   1:  PR[91,1] = PR[90,1] + 52.071;
   1:  PR[91,2] = PR[90,2] + -8.598;
   1:L PR[91] R[100]mm/sec CNT100;
   1:  PR[91,1] = PR[90,1] + 52.540;
   1:  PR[91,2] = PR[90,2] + -9.595;
   1:L PR[91] R[100]mm/sec CNT100;
   1:  PR[91,1] = PR[90,1] + 55.300;
   1:  PR[91,2] = PR[90,2] + -13.179;
   1:L PR[91] R[100]mm/sec CNT100;
   1:  PR[91,1] = PR[90,1] + 55.787;
   1:  PR[91,2] = PR[90,2] + -13.569;
   1:L PR[91] R[100]mm/sec CNT100;
   1:  PR[91,1] = PR[90,1] + 58.893;
   1:  PR[91,2] = PR[90,2] + -16.268;
   1:L PR[91] R[100]mm/sec CNT100;
   1:  PR[91,1] = PR[90,1] + 59.466;
   1:  PR[91,2] = PR[90,2] + -16.585;
   1:L PR[91] R[100]mm/sec CNT100;
   1:  PR[91,1] = PR[90,1] + 62.965;
   1:  PR[91,2] = PR[90,2] + -18.448;
   1:L PR[91] R[100]mm/sec CNT100;
   1:  PR[91,1] = PR[90,1] + 64.665;
   1:  PR[91,2] = PR[90,2] + -18.947;
   1:L PR[91] R[100]mm/sec CNT100;
   1:  PR[91,1] = PR[90,1] + 67.396;
   1:  PR[91,2] = PR[90,2] + -19.702;
   1:L PR[91] R[100]mm/sec CNT100;
   1:  PR[91,1] = PR[90,1] + 70.206;
   1:  PR[91,2] = PR[90,2] + -19.904;
   1:L PR[91] R[100]mm/sec CNT100;
   1:  PR[91,1] = PR[90,1] + 71.961;
   1:  PR[91,2] = PR[90,2] + -20.003;
   1:L PR[91] R[100]mm/sec CNT100;
   1:  PR[91,1] = PR[90,1] + 75.629;
   1:  PR[91,2] = PR[90,2] + -19.481;
   1:L PR[91] R[100]mm/sec CNT100;
   1:  PR[91,1] = PR[90,1] + 76.441;
   1:  PR[91,2] = PR[90,2] + -19.353;
   1:L PR[91] R[100]mm/sec CNT100;
   1:  PR[91,1] = PR[90,1] + 80.638;
   1:  PR[91,2] = PR[90,2] + -17.803;
   1:L PR[91] R[100]mm/sec CNT100;
   1:  PR[91,1] = PR[90,1] + 84.286;
   1:  PR[91,2] = PR[90,2] + -15.464;
   1:L PR[91] R[100]mm/sec CNT100;
   1:  PR[91,1] = PR[90,1] + 87.268;
   1:  PR[91,2] = PR[90,2] + -12.439;
   1:L PR[91] R[100]mm/sec CNT100TB   .50sec,CALL END_PUD;
   1:  PR[92] = PR[91];
   1:  PR[92,3] = PR[92,3] + 20;
   1:J PR[92] 10% FINE;
   1:  PR[91,1] = PR[90,1] + 39.000;
   1:  PR[91,2] = PR[90,2] + -12.973;
   1:  PR[92] = PR[91];
   1:  PR[92,3] = PR[92,3] + 20;
   1:J PR[92] 10% FINE;
   1:L PR[91] R[100]mm/sec CNT100;
   1:  CALL LASER_DRAHT_START;
   1:  PR[91,1] = PR[90,1] + 41.047;
   1:  PR[91,2] = PR[90,2] + -10.293;
   1:L PR[91] R[100]mm/sec CNT100;
   1:  PR[91,1] = PR[90,1] + 41.096;
   1:  PR[91,2] = PR[90,2] + -10.205;
   1:L PR[91] R[100]mm/sec CNT100;
   1:  PR[91,1] = PR[90,1] + 42.376;
   1:  PR[91,2] = PR[90,2] + -7.104;
   1:L PR[91] R[100]mm/sec CNT100;
   1:  PR[91,1] = PR[90,1] + 42.743;
   1:  PR[91,2] = PR[90,2] + -6.285;
   1:L PR[91] R[100]mm/sec CNT100;
   1:  PR[91,1] = PR[90,1] + 43.114;
   1:  PR[91,2] = PR[90,2] + -4.830;
   1:L PR[91] R[100]mm/sec CNT100;
   1:  PR[91,1] = PR[90,1] + 43.402;
   1:  PR[91,2] = PR[90,2] + -2.639;
   1:L PR[91] R[100]mm/sec CNT100;
   1:  PR[91,1] = PR[90,1] + 43.567;
   1:  PR[91,2] = PR[90,2] + -0.772;
   1:L PR[91] R[100]mm/sec CNT100;
   1:  PR[91,1] = PR[90,1] + 43.320;
   1:  PR[91,2] = PR[90,2] + 1.105;
   1:L PR[91] R[100]mm/sec CNT100;
   1:  PR[91,1] = PR[90,1] + 43.117;
   1:  PR[91,2] = PR[90,2] + 3.338;
   1:L PR[91] R[100]mm/sec CNT100;
   1:  PR[91,1] = PR[90,1] + 42.699;
   1:  PR[91,2] = PR[90,2] + 4.957;
   1:L PR[91] R[100]mm/sec CNT100;
   1:  PR[91,1] = PR[90,1] + 41.626;
   1:  PR[91,2] = PR[90,2] + 7.556;
   1:L PR[91] R[100]mm/sec CNT100;
   1:  PR[91,1] = PR[90,1] + 41.123;
   1:  PR[91,2] = PR[90,2] + 8.695;
   1:L PR[91] R[100]mm/sec CNT100;
   1:  PR[91,1] = PR[90,1] + 41.047;
   1:  PR[91,2] = PR[90,2] + 8.834;
   1:L PR[91] R[100]mm/sec CNT100;
   1:  PR[91,1] = PR[90,1] + 38.984;
   1:  PR[91,2] = PR[90,2] + 11.540;
   1:L PR[91] R[100]mm/sec CNT100;
   1:  PR[91,1] = PR[90,1] + 37.931;
   1:  PR[91,2] = PR[90,2] + 12.880;
   1:L PR[91] R[100]mm/sec CNT100;
   1:  PR[91,1] = PR[90,1] + 35.373;
   1:  PR[91,2] = PR[90,2] + 14.853;
   1:L PR[91] R[100]mm/sec CNT100;
   1:  PR[91,1] = PR[90,1] + 33.963;
   1:  PR[91,2] = PR[90,2] + 15.915;
   1:L PR[91] R[100]mm/sec CNT100;
   1:  PR[91,1] = PR[90,1] + 31.045;
   1:  PR[91,2] = PR[90,2] + 17.135;
   1:L PR[91] R[100]mm/sec CNT100;
   1:  PR[91,1] = PR[90,1] + 29.344;
   1:  PR[91,2] = PR[90,2] + 17.828;
   1:L PR[91] R[100]mm/sec CNT100;
   1:  PR[91,1] = PR[90,1] + 24.373;
   1:  PR[91,2] = PR[90,2] + 18.489;
   1:L PR[91] R[100]mm/sec CNT100;
   1:  PR[91,1] = PR[90,1] + 19.398;
   1:  PR[91,2] = PR[90,2] + 17.843;
   1:L PR[91] R[100]mm/sec CNT100;
   1:  PR[91,1] = PR[90,1] + 16.701;
   1:  PR[91,2] = PR[90,2] + 16.739;
   1:L PR[91] R[100]mm/sec CNT100;
   1:  PR[91,1] = PR[90,1] + 14.758;
   1:  PR[91,2] = PR[90,2] + 15.935;
   1:L PR[91] R[100]mm/sec CNT100;
   1:  PR[91,1] = PR[90,1] + 10.760;
   1:  PR[91,2] = PR[90,2] + 12.885;
   1:L PR[91] R[100]mm/sec CNT100;
   1:  PR[91,1] = PR[90,1] + 7.691;
   1:  PR[91,2] = PR[90,2] + 8.902;
   1:L PR[91] R[100]mm/sec CNT100;
   1:  PR[91,1] = PR[90,1] + 6.643;
   1:  PR[91,2] = PR[90,2] + 6.385;
   1:L PR[91] R[100]mm/sec CNT100;
   1:  PR[91,1] = PR[90,1] + 5.759;
   1:  PR[91,2] = PR[90,2] + 4.259;
   1:L PR[91] R[100]mm/sec CNT100;
   1:  PR[91,1] = PR[90,1] + 5.100;
   1:  PR[91,2] = PR[90,2] + -0.729;
   1:L PR[91] R[100]mm/sec CNT100;
   1:  PR[91,1] = PR[90,1] + 5.760;
   1:  PR[91,2] = PR[90,2] + -5.720;
   1:L PR[91] R[100]mm/sec CNT100;
   1:  PR[91,1] = PR[90,1] + 7.694;
   1:  PR[91,2] = PR[90,2] + -10.366;
   1:L PR[91] R[100]mm/sec CNT100;
   1:  PR[91,1] = PR[90,1] + 9.071;
   1:  PR[91,2] = PR[90,2] + -12.153;
   1:L PR[91] R[100]mm/sec CNT100;
   1:  PR[91,1] = PR[90,1] + 10.765;
   1:  PR[91,2] = PR[90,2] + -14.349;
   1:L PR[91] R[100]mm/sec CNT100;
   1:  PR[91,1] = PR[90,1] + 14.764;
   1:  PR[91,2] = PR[90,2] + -17.397;
   1:L PR[91] R[100]mm/sec CNT100;
   1:  PR[91,1] = PR[90,1] + 19.412;
   1:  PR[91,2] = PR[90,2] + -19.306;
   1:L PR[91] R[100]mm/sec CNT100;
   1:  PR[91,1] = PR[90,1] + 21.410;
   1:  PR[91,2] = PR[90,2] + -19.568;
   1:L PR[91] R[100]mm/sec CNT100;
   1:  PR[91,1] = PR[90,1] + 24.384;
   1:  PR[91,2] = PR[90,2] + -19.948;
   1:L PR[91] R[100]mm/sec CNT100;
   1:  PR[91,1] = PR[90,1] + 29.352;
   1:  PR[91,2] = PR[90,2] + -19.284;
   1:L PR[91] R[100]mm/sec CNT100;
   1:  PR[91,1] = PR[90,1] + 33.978;
   1:  PR[91,2] = PR[90,2] + -17.364;
   1:L PR[91] R[100]mm/sec CNT100;
   1:  PR[91,1] = PR[90,1] + 35.384;
   1:  PR[91,2] = PR[90,2] + -16.300;
   1:L PR[91] R[100]mm/sec CNT100;
   1:  PR[91,1] = PR[90,1] + 37.942;
   1:  PR[91,2] = PR[90,2] + -14.327;
   1:L PR[91] R[100]mm/sec CNT100;
   1:  PR[91,1] = PR[90,1] + 39.000;
   1:  PR[91,2] = PR[90,2] + -12.973;
   1:L PR[91] R[100]mm/sec CNT100TB   .50sec,CALL END_PUD;
   1:  PR[92] = PR[91];
   1:  PR[92,3] = PR[92,3] + 20;
   1:J PR[92] 10% FINE;
   1:  PR[91,1] = PR[90,1] + -35.031;
   1:  PR[91,2] = PR[90,2] + -15.307;
   1:  PR[92] = PR[91];
   1:  PR[92,3] = PR[92,3] + 20;
   1:J PR[92] 10% FINE;
   1:L PR[91] R[100]mm/sec CNT100;
   1:  CALL LASER_DRAHT_START;
   1:  PR[91,1] = PR[90,1] + -31.479;
   1:  PR[91,2] = PR[90,2] + -17.570;
   1:L PR[91] R[100]mm/sec CNT100;
   1:  PR[91,1] = PR[90,1] + -29.846;
   1:  PR[91,2] = PR[90,2] + -18.148;
   1:L PR[91] R[100]mm/sec CNT100;
   1:  PR[91,1] = PR[90,1] + -27.490;
   1:  PR[91,2] = PR[90,2] + -19.008;
   1:L PR[91] R[100]mm/sec CNT100;
   1:  PR[91,1] = PR[90,1] + -26.011;
   1:  PR[91,2] = PR[90,2] + -19.184;
   1:L PR[91] R[100]mm/sec CNT100;
   1:  PR[91,1] = PR[90,1] + -23.269;
   1:  PR[91,2] = PR[90,2] + -19.541;
   1:L PR[91] R[100]mm/sec CNT100;
   1:  PR[91,1] = PR[90,1] + -22.057;
   1:  PR[91,2] = PR[90,2] + -19.415;
   1:L PR[91] R[100]mm/sec CNT100;
   1:  PR[91,1] = PR[90,1] + -19.010;
   1:  PR[91,2] = PR[90,2] + -19.132;
   1:L PR[91] R[100]mm/sec CNT100;
   1:  PR[91,1] = PR[90,1] + -14.945;
   1:  PR[91,2] = PR[90,2] + -17.797;
   1:L PR[91] R[100]mm/sec CNT100;
   1:  PR[91,1] = PR[90,1] + -11.270;
   1:  PR[91,2] = PR[90,2] + -15.588;
   1:L PR[91] R[100]mm/sec CNT100;
   1:  PR[91,1] = PR[90,1] + -8.180;
   1:  PR[91,2] = PR[90,2] + -12.612;
   1:L PR[91] R[100]mm/sec CNT100;
   1:  PR[91,1] = PR[90,1] + -5.841;
   1:  PR[91,2] = PR[90,2] + -9.017;
   1:L PR[91] R[100]mm/sec CNT100;
   1:  PR[91,1] = PR[90,1] + -4.786;
   1:  PR[91,2] = PR[90,2] + -6.096;
   1:L PR[91] R[100]mm/sec CNT100;
   1:  PR[91,1] = PR[90,1] + -4.371;
   1:  PR[91,2] = PR[90,2] + -4.985;
   1:L PR[91] R[100]mm/sec CNT100;
   1:  PR[91,1] = PR[90,1] + -3.858;
   1:  PR[91,2] = PR[90,2] + -0.763;
   1:L PR[91] R[100]mm/sec CNT100;
   1:  PR[91,1] = PR[90,1] + -4.364;
   1:  PR[91,2] = PR[90,2] + 3.490;
   1:L PR[91] R[100]mm/sec CNT100;
   1:  PR[91,1] = PR[90,1] + -5.841;
   1:  PR[91,2] = PR[90,2] + 7.557;
   1:L PR[91] R[100]mm/sec CNT100;
   1:  PR[91,1] = PR[90,1] + -8.180;
   1:  PR[91,2] = PR[90,2] + 11.154;
   1:L PR[91] R[100]mm/sec CNT100;
   1:  PR[91,1] = PR[90,1] + -11.276;
   1:  PR[91,2] = PR[90,2] + 14.134;
   1:L PR[91] R[100]mm/sec CNT100;
   1:  PR[91,1] = PR[90,1] + -11.596;
   1:  PR[91,2] = PR[90,2] + 14.330;
   1:L PR[91] R[100]mm/sec CNT100;
   1:  PR[91,1] = PR[90,1] + -14.944;
   1:  PR[91,2] = PR[90,2] + 16.337;
   1:L PR[91] R[100]mm/sec CNT100;
   1:  PR[91,1] = PR[90,1] + -19.013;
   1:  PR[91,2] = PR[90,2] + 17.674;
   1:L PR[91] R[100]mm/sec CNT100;
   1:  PR[91,1] = PR[90,1] + -23.265;
   1:  PR[91,2] = PR[90,2] + 18.084;
   1:L PR[91] R[100]mm/sec CNT100;
   1:  PR[91,1] = PR[90,1] + -27.488;
   1:  PR[91,2] = PR[90,2] + 17.551;
   1:L PR[91] R[100]mm/sec CNT100;
   1:  PR[91,1] = PR[90,1] + -31.478;
   1:  PR[91,2] = PR[90,2] + 16.113;
   1:L PR[91] R[100]mm/sec CNT100;
   1:  PR[91,1] = PR[90,1] + -33.041;
   1:  PR[91,2] = PR[90,2] + 15.126;
   1:L PR[91] R[100]mm/sec CNT100;
   1:  PR[91,1] = PR[90,1] + -35.028;
   1:  PR[91,2] = PR[90,2] + 13.851;
   1:L PR[91] R[100]mm/sec CNT100;
   1:  PR[91,1] = PR[90,1] + -37.988;
   1:  PR[91,2] = PR[90,2] + 10.872;
   1:L PR[91] R[100]mm/sec CNT100;
   1:  PR[91,1] = PR[90,1] + -40.205;
   1:  PR[91,2] = PR[90,2] + 7.331;
   1:L PR[91] R[100]mm/sec CNT100;
   1:  PR[91,1] = PR[90,1] + -41.577;
   1:  PR[91,2] = PR[90,2] + 3.400;
   1:L PR[91] R[100]mm/sec CNT100;
   1:  PR[91,1] = PR[90,1] + -41.851;
   1:  PR[91,2] = PR[90,2] + 0.989;
   1:L PR[91] R[100]mm/sec CNT100;
   1:  PR[91,1] = PR[90,1] + -41.912;
   1:  PR[91,2] = PR[90,2] + 0.689;
   1:L PR[91] R[100]mm/sec CNT100;
   1:  PR[91,1] = PR[90,1] + -42.070;
   1:  PR[91,2] = PR[90,2] + -0.717;
   1:L PR[91] R[100]mm/sec CNT100;
   1:  PR[91,1] = PR[90,1] + -41.780;
   1:  PR[91,2] = PR[90,2] + -3.046;
   1:L PR[91] R[100]mm/sec CNT100;
   1:  PR[91,1] = PR[90,1] + -41.577;
   1:  PR[91,2] = PR[90,2] + -4.860;
   1:L PR[91] R[100]mm/sec CNT100;
   1:  PR[91,1] = PR[90,1] + -40.205;
   1:  PR[91,2] = PR[90,2] + -8.790;
   1:L PR[91] R[100]mm/sec CNT100;
   1:  PR[91,1] = PR[90,1] + -37.988;
   1:  PR[91,2] = PR[90,2] + -12.331;
   1:L PR[91] R[100]mm/sec CNT100;
   1:  PR[91,1] = PR[90,1] + -35.031;
   1:  PR[91,2] = PR[90,2] + -15.307;
   1:L PR[91] R[100]mm/sec CNT100TB   .50sec,CALL END_PUD;
   1:  PR[92] = PR[91];
   1:  PR[92,3] = PR[92,3] + 20;
   1:J PR[92] 10% FINE;
   1:  PR[91,1] = PR[90,1] + -52.444;
   1:  PR[91,2] = PR[90,2] + -4.731;
   1:  PR[92] = PR[91];
   1:  PR[92,3] = PR[92,3] + 20;
   1:J PR[92] 10% FINE;
   1:L PR[91] R[100]mm/sec CNT100;
   1:  CALL LASER_DRAHT_START;
   1:  PR[91,1] = PR[90,1] + -52.394;
   1:  PR[91,2] = PR[90,2] + -4.297;
   1:L PR[91] R[100]mm/sec CNT100;
   1:  PR[91,1] = PR[90,1] + -52.278;
   1:  PR[91,2] = PR[90,2] + -2.705;
   1:L PR[91] R[100]mm/sec CNT100;
   1:  PR[91,1] = PR[90,1] + -52.049;
   1:  PR[91,2] = PR[90,2] + -0.729;
   1:L PR[91] R[100]mm/sec CNT100;
   1:  PR[91,1] = PR[90,1] + -52.298;
   1:  PR[91,2] = PR[90,2] + 1.418;
   1:L PR[91] R[100]mm/sec CNT100;
   1:  PR[91,1] = PR[90,1] + -52.415;
   1:  PR[91,2] = PR[90,2] + 2.813;
   1:L PR[91] R[100]mm/sec CNT100;
   1:  PR[91,1] = PR[90,1] + -52.468;
   1:  PR[91,2] = PR[90,2] + 3.254;
   1:L PR[91] R[100]mm/sec CNT100;
   1:  PR[91,1] = PR[90,1] + -53.877;
   1:  PR[91,2] = PR[90,2] + 7.045;
   1:L PR[91] R[100]mm/sec CNT100;
   1:  PR[91,1] = PR[90,1] + -55.077;
   1:  PR[91,2] = PR[90,2] + 8.853;
   1:L PR[91] R[100]mm/sec CNT100;
   1:  PR[91,1] = PR[90,1] + -56.120;
   1:  PR[91,2] = PR[90,2] + 10.513;
   1:L PR[91] R[100]mm/sec CNT100;
   1:  PR[91,1] = PR[90,1] + -58.984;
   1:  PR[91,2] = PR[90,2] + 13.425;
   1:L PR[91] R[100]mm/sec CNT100;
   1:  PR[91,1] = PR[90,1] + -62.416;
   1:  PR[91,2] = PR[90,2] + 15.689;
   1:L PR[91] R[100]mm/sec CNT100;
   1:  PR[91,1] = PR[90,1] + -63.818;
   1:  PR[91,2] = PR[90,2] + 16.256;
   1:L PR[91] R[100]mm/sec CNT100;
   1:  PR[91,1] = PR[90,1] + -66.237;
   1:  PR[91,2] = PR[90,2] + 17.207;
   1:L PR[91] R[100]mm/sec CNT100;
   1:  PR[91,1] = PR[90,1] + -68.485;
   1:  PR[91,2] = PR[90,2] + 17.619;
   1:L PR[91] R[100]mm/sec CNT100;
   1:  PR[91,1] = PR[90,1] + -70.282;
   1:  PR[91,2] = PR[90,2] + 17.931;
   1:L PR[91] R[100]mm/sec CNT100;
   1:  PR[91,1] = PR[90,1] + -74.386;
   1:  PR[91,2] = PR[90,2] + 17.839;
   1:L PR[91] R[100]mm/sec CNT100;
   1:  PR[91,1] = PR[90,1] + -78.357;
   1:  PR[91,2] = PR[90,2] + 16.946;
   1:L PR[91] R[100]mm/sec CNT100;
   1:  PR[91,1] = PR[90,1] + -82.028;
   1:  PR[91,2] = PR[90,2] + 15.300;
   1:L PR[91] R[100]mm/sec CNT100;
   1:  PR[91,1] = PR[90,1] + -85.206;
   1:  PR[91,2] = PR[90,2] + 12.990;
   1:L PR[91] R[100]mm/sec CNT100;
   1:  PR[91,1] = PR[90,1] + -87.798;
   1:  PR[91,2] = PR[90,2] + 10.103;
   1:L PR[91] R[100]mm/sec CNT100;
   1:  PR[91,1] = PR[90,1] + -89.732;
   1:  PR[91,2] = PR[90,2] + 6.757;
   1:L PR[91] R[100]mm/sec CNT100;
   1:  PR[91,1] = PR[90,1] + -90.923;
   1:  PR[91,2] = PR[90,2] + 3.093;
   1:L PR[91] R[100]mm/sec CNT100;
   1:  PR[91,1] = PR[90,1] + -90.982;
   1:  PR[91,2] = PR[90,2] + 2.544;
   1:L PR[91] R[100]mm/sec CNT100;
   1:  PR[91,1] = PR[90,1] + -91.135;
   1:  PR[91,2] = PR[90,2] + 1.574;
   1:L PR[91] R[100]mm/sec CNT100;
   1:  PR[91,1] = PR[90,1] + -91.373;
   1:  PR[91,2] = PR[90,2] + -0.678;
   1:L PR[91] R[100]mm/sec CNT100;
   1:  PR[91,1] = PR[90,1] + -91.293;
   1:  PR[91,2] = PR[90,2] + -1.188;
   1:L PR[91] R[100]mm/sec CNT100;
   1:  PR[91,1] = PR[90,1] + -91.126;
   1:  PR[91,2] = PR[90,2] + -1.902;
   1:L PR[91] R[100]mm/sec CNT100;
   1:  PR[91,1] = PR[90,1] + -90.848;
   1:  PR[91,2] = PR[90,2] + -4.554;
   1:L PR[91] R[100]mm/sec CNT100;
   1:  PR[91,1] = PR[90,1] + -90.460;
   1:  PR[91,2] = PR[90,2] + -5.739;
   1:L PR[91] R[100]mm/sec CNT100;
   1:  PR[91,1] = PR[90,1] + -89.653;
   1:  PR[91,2] = PR[90,2] + -8.221;
   1:L PR[91] R[100]mm/sec CNT100;
   1:  PR[91,1] = PR[90,1] + -87.714;
   1:  PR[91,2] = PR[90,2] + -11.570;
   1:L PR[91] R[100]mm/sec CNT100;
   1:  PR[91,1] = PR[90,1] + -85.111;
   1:  PR[91,2] = PR[90,2] + -14.465;
   1:L PR[91] R[100]mm/sec CNT100;
   1:  PR[91,1] = PR[90,1] + -81.948;
   1:  PR[91,2] = PR[90,2] + -16.777;
   1:L PR[91] R[100]mm/sec CNT100;
   1:  PR[91,1] = PR[90,1] + -78.359;
   1:  PR[91,2] = PR[90,2] + -18.406;
   1:L PR[91] R[100]mm/sec CNT100;
   1:  PR[91,1] = PR[90,1] + -74.469;
   1:  PR[91,2] = PR[90,2] + -19.281;
   1:L PR[91] R[100]mm/sec CNT100;
   1:  PR[91,1] = PR[90,1] + -70.334;
   1:  PR[91,2] = PR[90,2] + -19.379;
   1:L PR[91] R[100]mm/sec CNT100;
   1:  PR[91,1] = PR[90,1] + -67.041;
   1:  PR[91,2] = PR[90,2] + -18.790;
   1:L PR[91] R[100]mm/sec CNT100;
   1:  PR[91,1] = PR[90,1] + -66.230;
   1:  PR[91,2] = PR[90,2] + -18.657;
   1:L PR[91] R[100]mm/sec CNT100;
   1:  PR[91,1] = PR[90,1] + -63.633;
   1:  PR[91,2] = PR[90,2] + -17.624;
   1:L PR[91] R[100]mm/sec CNT100;
   1:  PR[91,1] = PR[90,1] + -62.365;
   1:  PR[91,2] = PR[90,2] + -17.142;
   1:L PR[91] R[100]mm/sec CNT100;
   1:  PR[91,1] = PR[90,1] + -60.499;
   1:  PR[91,2] = PR[90,2] + -15.910;
   1:L PR[91] R[100]mm/sec CNT100;
   1:  PR[91,1] = PR[90,1] + -58.899;
   1:  PR[91,2] = PR[90,2] + -14.886;
   1:L PR[91] R[100]mm/sec CNT100;
   1:  PR[91,1] = PR[90,1] + -57.721;
   1:  PR[91,2] = PR[90,2] + -13.686;
   1:L PR[91] R[100]mm/sec CNT100;
   1:  PR[91,1] = PR[90,1] + -55.994;
   1:  PR[91,2] = PR[90,2] + -11.972;
   1:L PR[91] R[100]mm/sec CNT100;
   1:  PR[91,1] = PR[90,1] + -53.806;
   1:  PR[91,2] = PR[90,2] + -8.540;
   1:L PR[91] R[100]mm/sec CNT100;
   1:  PR[91,1] = PR[90,1] + -52.444;
   1:  PR[91,2] = PR[90,2] + -4.731;
   1:L PR[91] R[100]mm/sec CNT100TB   .50sec,CALL END_PUD;
   1:  PR[92] = PR[91];
   1:  PR[92,3] = PR[92,3] + 20;
   1:J PR[92] 10% FINE;
   1:  PR[91] = PR[90];
   1:  PR[91,1] = PR[90,1] + 65.665;
   1:  PR[91,2] = PR[90,2] + 18.026;
   1:  PR[91,3] = PR[90,3] + 30.095;
   1:  PR[92] = PR[91];
   1:  PR[92,3] = PR[92,3] + 20;
   1:J PR[92] 10% FINE;
   1:L PR[91] R[100]mm/sec CNT100;
   1:  CALL LASER_DRAHT_START;
   1:  PR[91,1] = PR[90,1] + 62.481;
   1:  PR[91,2] = PR[90,2] + 17.159;
   1:L PR[91] R[100]mm/sec CNT100;
   1:  PR[91,1] = PR[90,1] + 62.045;
   1:  PR[91,2] = PR[90,2] + 16.917;
   1:L PR[91] R[100]mm/sec CNT100;
   1:  PR[91,1] = PR[90,1] + 58.910;
   1:  PR[91,2] = PR[90,2] + 15.262;
   1:L PR[91] R[100]mm/sec CNT100;
   1:  PR[91,1] = PR[90,1] + 58.234;
   1:  PR[91,2] = PR[90,2] + 14.935;
   1:L PR[91] R[100]mm/sec CNT100;
   1:  PR[91,1] = PR[90,1] + 58.180;
   1:  PR[91,2] = PR[90,2] + 14.897;
   1:L PR[91] R[100]mm/sec CNT100;
   1:  PR[91,1] = PR[90,1] + 54.683;
   1:  PR[91,2] = PR[90,2] + 12.095;
   1:L PR[91] R[100]mm/sec CNT100;
   1:  PR[91,1] = PR[90,1] + 53.674;
   1:  PR[91,2] = PR[90,2] + 10.924;
   1:L PR[91] R[100]mm/sec CNT100;
   1:  PR[91,1] = PR[90,1] + 51.769;
   1:  PR[91,2] = PR[90,2] + 8.450;
   1:L PR[91] R[100]mm/sec CNT100;
   1:  PR[91,1] = PR[90,1] + 50.629;
   1:  PR[91,2] = PR[90,2] + 6.027;
   1:L PR[91] R[100]mm/sec CNT100;
   1:  PR[91,1] = PR[90,1] + 49.813;
   1:  PR[91,2] = PR[90,2] + 4.103;
   1:L PR[91] R[100]mm/sec CNT100;
   1:  PR[91,1] = PR[90,1] + 49.326;
   1:  PR[91,2] = PR[90,2] + 0.913;
   1:L PR[91] R[100]mm/sec CNT100;
   1:  PR[91,1] = PR[90,1] + 49.102;
   1:  PR[91,2] = PR[90,2] + -0.695;
   1:L PR[91] R[100]mm/sec CNT100;
   1:  PR[91,1] = PR[90,1] + 49.327;
   1:  PR[91,2] = PR[90,2] + -2.379;
   1:L PR[91] R[100]mm/sec CNT100;
   1:  PR[91,1] = PR[90,1] + 49.813;
   1:  PR[91,2] = PR[90,2] + -5.561;
   1:L PR[91] R[100]mm/sec CNT100;
   1:  PR[91,1] = PR[90,1] + 50.629;
   1:  PR[91,2] = PR[90,2] + -7.485;
   1:L PR[91] R[100]mm/sec CNT100;
   1:  PR[91,1] = PR[90,1] + 51.768;
   1:  PR[91,2] = PR[90,2] + -9.909;
   1:L PR[91] R[100]mm/sec CNT100;
   1:  PR[91,1] = PR[90,1] + 53.673;
   1:  PR[91,2] = PR[90,2] + -12.382;
   1:L PR[91] R[100]mm/sec CNT100;
   1:  PR[91,1] = PR[90,1] + 54.682;
   1:  PR[91,2] = PR[90,2] + -13.554;
   1:L PR[91] R[100]mm/sec CNT100;
   1:  PR[91,1] = PR[90,1] + 58.180;
   1:  PR[91,2] = PR[90,2] + -16.356;
   1:L PR[91] R[100]mm/sec CNT100;
   1:  PR[91,1] = PR[90,1] + 58.234;
   1:  PR[91,2] = PR[90,2] + -16.393;
   1:L PR[91] R[100]mm/sec CNT100;
   1:  PR[91,1] = PR[90,1] + 58.913;
   1:  PR[91,2] = PR[90,2] + -16.723;
   1:L PR[91] R[100]mm/sec CNT100;
   1:  PR[91,1] = PR[90,1] + 62.480;
   1:  PR[91,2] = PR[90,2] + -18.622;
   1:L PR[91] R[100]mm/sec CNT100;
   1:  PR[91,1] = PR[90,1] + 63.191;
   1:  PR[91,2] = PR[90,2] + -18.831;
   1:L PR[91] R[100]mm/sec CNT100;
   1:  PR[91,1] = PR[90,1] + 66.959;
   1:  PR[91,2] = PR[90,2] + -19.873;
   1:L PR[91] R[100]mm/sec CNT100;
   1:  PR[91,1] = PR[90,1] + 68.821;
   1:  PR[91,2] = PR[90,2] + -20.006;
   1:L PR[91] R[100]mm/sec CNT100;
   1:  PR[91,1] = PR[90,1] + 71.564;
   1:  PR[91,2] = PR[90,2] + -20.161;
   1:L PR[91] R[100]mm/sec CNT100;
   1:  PR[91,1] = PR[90,1] + 74.370;
   1:  PR[91,2] = PR[90,2] + -19.761;
   1:L PR[91] R[100]mm/sec CNT100;
   1:  PR[91,1] = PR[90,1] + 76.078;
   1:  PR[91,2] = PR[90,2] + -19.494;
   1:L PR[91] R[100]mm/sec CNT100;
   1:  PR[91,1] = PR[90,1] + 79.461;
   1:  PR[91,2] = PR[90,2] + -18.247;
   1:L PR[91] R[100]mm/sec CNT100;
   1:  PR[91,1] = PR[90,1] + 80.291;
   1:  PR[91,2] = PR[90,2] + -17.928;
   1:L PR[91] R[100]mm/sec CNT100;
   1:  PR[91,1] = PR[90,1] + 84.027;
   1:  PR[91,2] = PR[90,2] + -15.542;
   1:L PR[91] R[100]mm/sec CNT100;
   1:  PR[91,1] = PR[90,1] + 87.096;
   1:  PR[91,2] = PR[90,2] + -12.480;
   1:L PR[91] R[100]mm/sec CNT100;
   1:  PR[91,1] = PR[90,1] + 89.333;
   1:  PR[91,2] = PR[90,2] + -8.889;
   1:L PR[91] R[100]mm/sec CNT100;
   1:  PR[91,1] = PR[90,1] + 90.726;
   1:  PR[91,2] = PR[90,2] + -4.882;
   1:L PR[91] R[100]mm/sec CNT100;
   1:  PR[91,1] = PR[90,1] + 90.839;
   1:  PR[91,2] = PR[90,2] + -4.069;
   1:L PR[91] R[100]mm/sec CNT100;
   1:  PR[91,1] = PR[90,1] + 91.206;
   1:  PR[91,2] = PR[90,2] + -0.801;
   1:L PR[91] R[100]mm/sec CNT100;
   1:  PR[91,1] = PR[90,1] + 91.161;
   1:  PR[91,2] = PR[90,2] + -0.555;
   1:L PR[91] R[100]mm/sec CNT100;
   1:  PR[91,1] = PR[90,1] + 90.717;
   1:  PR[91,2] = PR[90,2] + 3.449;
   1:L PR[91] R[100]mm/sec CNT100;
   1:  PR[91,1] = PR[90,1] + 89.333;
   1:  PR[91,2] = PR[90,2] + 7.430;
   1:L PR[91] R[100]mm/sec CNT100;
   1:  PR[91,1] = PR[90,1] + 87.096;
   1:  PR[91,2] = PR[90,2] + 11.022;
   1:L PR[91] R[100]mm/sec CNT100;
   1:  PR[91,1] = PR[90,1] + 84.027;
   1:  PR[91,2] = PR[90,2] + 14.083;
   1:L PR[91] R[100]mm/sec CNT100;
   1:  PR[91,1] = PR[90,1] + 80.304;
   1:  PR[91,2] = PR[90,2] + 16.461;
   1:L PR[91] R[100]mm/sec CNT100;
   1:  PR[91,1] = PR[90,1] + 77.126;
   1:  PR[91,2] = PR[90,2] + 17.626;
   1:L PR[91] R[100]mm/sec CNT100;
   1:  PR[91,1] = PR[90,1] + 76.078;
   1:  PR[91,2] = PR[90,2] + 18.031;
   1:L PR[91] R[100]mm/sec CNT100;
   1:  PR[91,1] = PR[90,1] + 73.304;
   1:  PR[91,2] = PR[90,2] + 18.419;
   1:L PR[91] R[100]mm/sec CNT100;
   1:  PR[91,1] = PR[90,1] + 71.564;
   1:  PR[91,2] = PR[90,2] + 18.698;
   1:L PR[91] R[100]mm/sec CNT100;
   1:  PR[91,1] = PR[90,1] + 69.448;
   1:  PR[91,2] = PR[90,2] + 18.541;
   1:L PR[91] R[100]mm/sec CNT100;
   1:  PR[91,1] = PR[90,1] + 66.959;
   1:  PR[91,2] = PR[90,2] + 18.410;
   1:L PR[91] R[100]mm/sec CNT100;
   1:  PR[91,1] = PR[90,1] + 65.665;
   1:  PR[91,2] = PR[90,2] + 18.026;
   1:L PR[91] R[100]mm/sec CNT100TB   .50sec,CALL END_PUD;
   1:  PR[92] = PR[91];
   1:  PR[92,3] = PR[92,3] + 20;
   1:J PR[92] 10% FINE;
   1:  PR[91,1] = PR[90,1] + 42.274;
   1:  PR[91,2] = PR[90,2] + -7.577;
   1:  PR[92] = PR[91];
   1:  PR[92,3] = PR[92,3] + 20;
   1:J PR[92] 10% FINE;
   1:L PR[91] R[100]mm/sec CNT100;
   1:  CALL LASER_DRAHT_START;
   1:  PR[91,1] = PR[90,1] + 42.750;
   1:  PR[91,2] = PR[90,2] + -6.514;
   1:L PR[91] R[100]mm/sec CNT100;
   1:  PR[91,1] = PR[90,1] + 43.237;
   1:  PR[91,2] = PR[90,2] + -4.609;
   1:L PR[91] R[100]mm/sec CNT100;
   1:  PR[91,1] = PR[90,1] + 43.424;
   1:  PR[91,2] = PR[90,2] + -3.188;
   1:L PR[91] R[100]mm/sec CNT100;
   1:  PR[91,1] = PR[90,1] + 43.637;
   1:  PR[91,2] = PR[90,2] + -0.772;
   1:L PR[91] R[100]mm/sec CNT100;
   1:  PR[91,1] = PR[90,1] + 43.502;
   1:  PR[91,2] = PR[90,2] + 0.258;
   1:L PR[91] R[100]mm/sec CNT100;
   1:  PR[91,1] = PR[90,1] + 43.243;
   1:  PR[91,2] = PR[90,2] + 3.100;
   1:L PR[91] R[100]mm/sec CNT100;
   1:  PR[91,1] = PR[90,1] + 42.697;
   1:  PR[91,2] = PR[90,2] + 5.213;
   1:L PR[91] R[100]mm/sec CNT100;
   1:  PR[91,1] = PR[90,1] + 41.859;
   1:  PR[91,2] = PR[90,2] + 7.242;
   1:L PR[91] R[100]mm/sec CNT100;
   1:  PR[91,1] = PR[90,1] + 41.217;
   1:  PR[91,2] = PR[90,2] + 8.697;
   1:L PR[91] R[100]mm/sec CNT100;
   1:  PR[91,1] = PR[90,1] + 41.093;
   1:  PR[91,2] = PR[90,2] + 8.924;
   1:L PR[91] R[100]mm/sec CNT100;
   1:  PR[91,1] = PR[90,1] + 39.306;
   1:  PR[91,2] = PR[90,2] + 11.270;
   1:L PR[91] R[100]mm/sec CNT100;
   1:  PR[91,1] = PR[90,1] + 37.948;
   1:  PR[91,2] = PR[90,2] + 12.997;
   1:L PR[91] R[100]mm/sec CNT100;
   1:  PR[91,1] = PR[90,1] + 35.756;
   1:  PR[91,2] = PR[90,2] + 14.688;
   1:L PR[91] R[100]mm/sec CNT100;
   1:  PR[91,1] = PR[90,1] + 33.951;
   1:  PR[91,2] = PR[90,2] + 16.047;
   1:L PR[91] R[100]mm/sec CNT100;
   1:  PR[91,1] = PR[90,1] + 31.464;
   1:  PR[91,2] = PR[90,2] + 17.087;
   1:L PR[91] R[100]mm/sec CNT100;
   1:  PR[91,1] = PR[90,1] + 29.300;
   1:  PR[91,2] = PR[90,2] + 17.969;
   1:L PR[91] R[100]mm/sec CNT100;
   1:  PR[91,1] = PR[90,1] + 24.296;
   1:  PR[91,2] = PR[90,2] + 18.631;
   1:L PR[91] R[100]mm/sec CNT100;
   1:  PR[91,1] = PR[90,1] + 19.286;
   1:  PR[91,2] = PR[90,2] + 17.979;
   1:L PR[91] R[100]mm/sec CNT100;
   1:  PR[91,1] = PR[90,1] + 17.035;
   1:  PR[91,2] = PR[90,2] + 17.057;
   1:L PR[91] R[100]mm/sec CNT100;
   1:  PR[91,1] = PR[90,1] + 14.614;
   1:  PR[91,2] = PR[90,2] + 16.055;
   1:L PR[91] R[100]mm/sec CNT100;
   1:  PR[91,1] = PR[90,1] + 10.590;
   1:  PR[91,2] = PR[90,2] + 12.984;
   1:L PR[91] R[100]mm/sec CNT100;
   1:  PR[91,1] = PR[90,1] + 7.499;
   1:  PR[91,2] = PR[90,2] + 8.972;
   1:L PR[91] R[100]mm/sec CNT100;
   1:  PR[91,1] = PR[90,1] + 6.643;
   1:  PR[91,2] = PR[90,2] + 6.918;
   1:L PR[91] R[100]mm/sec CNT100;
   1:  PR[91,1] = PR[90,1] + 5.553;
   1:  PR[91,2] = PR[90,2] + 4.295;
   1:L PR[91] R[100]mm/sec CNT100;
   1:  PR[91,1] = PR[90,1] + 4.889;
   1:  PR[91,2] = PR[90,2] + -0.729;
   1:L PR[91] R[100]mm/sec CNT100;
   1:  PR[91,1] = PR[90,1] + 5.554;
   1:  PR[91,2] = PR[90,2] + -5.756;
   1:L PR[91] R[100]mm/sec CNT100;
   1:  PR[91,1] = PR[90,1] + 7.502;
   1:  PR[91,2] = PR[90,2] + -10.436;
   1:L PR[91] R[100]mm/sec CNT100;
   1:  PR[91,1] = PR[90,1] + 9.203;
   1:  PR[91,2] = PR[90,2] + -12.645;
   1:L PR[91] R[100]mm/sec CNT100;
   1:  PR[91,1] = PR[90,1] + 10.595;
   1:  PR[91,2] = PR[90,2] + -14.448;
   1:L PR[91] R[100]mm/sec CNT100;
   1:  PR[91,1] = PR[90,1] + 14.622;
   1:  PR[91,2] = PR[90,2] + -17.519;
   1:L PR[91] R[100]mm/sec CNT100;
   1:  PR[91,1] = PR[90,1] + 19.303;
   1:  PR[91,2] = PR[90,2] + -19.442;
   1:L PR[91] R[100]mm/sec CNT100;
   1:  PR[91,1] = PR[90,1] + 21.809;
   1:  PR[91,2] = PR[90,2] + -19.771;
   1:L PR[91] R[100]mm/sec CNT100;
   1:  PR[91,1] = PR[90,1] + 24.309;
   1:  PR[91,2] = PR[90,2] + -20.090;
   1:L PR[91] R[100]mm/sec CNT100;
   1:  PR[91,1] = PR[90,1] + 29.312;
   1:  PR[91,2] = PR[90,2] + -19.424;
   1:L PR[91] R[100]mm/sec CNT100;
   1:  PR[91,1] = PR[90,1] + 33.970;
   1:  PR[91,2] = PR[90,2] + -17.495;
   1:L PR[91] R[100]mm/sec CNT100;
   1:  PR[91,1] = PR[90,1] + 35.771;
   1:  PR[91,2] = PR[90,2] + -16.131;
   1:L PR[91] R[100]mm/sec CNT100;
   1:  PR[91,1] = PR[90,1] + 37.962;
   1:  PR[91,2] = PR[90,2] + -14.441;
   1:L PR[91] R[100]mm/sec CNT100;
   1:  PR[91,1] = PR[90,1] + 39.326;
   1:  PR[91,2] = PR[90,2] + -12.696;
   1:L PR[91] R[100]mm/sec CNT100;
   1:  PR[91,1] = PR[90,1] + 41.093;
   1:  PR[91,2] = PR[90,2] + -10.384;
   1:L PR[91] R[100]mm/sec CNT100;
   1:  PR[91,1] = PR[90,1] + 41.185;
   1:  PR[91,2] = PR[90,2] + -10.215;
   1:L PR[91] R[100]mm/sec CNT100;
   1:  PR[91,1] = PR[90,1] + 42.274;
   1:  PR[91,2] = PR[90,2] + -7.577;
   1:L PR[91] R[100]mm/sec CNT100TB   .50sec,CALL END_PUD;
   1:  PR[92] = PR[91];
   1:  PR[92,3] = PR[92,3] + 20;
   1:J PR[92] 10% FINE;
   1:  PR[91,1] = PR[90,1] + -5.269;
   1:  PR[91,2] = PR[90,2] + 7.364;
   1:  PR[92] = PR[91];
   1:  PR[92,3] = PR[92,3] + 20;
   1:J PR[92] 10% FINE;
   1:L PR[91] R[100]mm/sec CNT100;
   1:  CALL LASER_DRAHT_START;
   1:  PR[91,1] = PR[90,1] + -5.412;
   1:  PR[91,2] = PR[90,2] + 7.679;
   1:L PR[91] R[100]mm/sec CNT100;
   1:  PR[91,1] = PR[90,1] + -7.750;
   1:  PR[91,2] = PR[90,2] + 11.155;
   1:L PR[91] R[100]mm/sec CNT100;
   1:  PR[91,1] = PR[90,1] + -7.803;
   1:  PR[91,2] = PR[90,2] + 11.224;
   1:L PR[91] R[100]mm/sec CNT100;
   1:  PR[91,1] = PR[90,1] + -10.999;
   1:  PR[91,2] = PR[90,2] + 14.200;
   1:L PR[91] R[100]mm/sec CNT100;
   1:  PR[91,1] = PR[90,1] + -14.709;
   1:  PR[91,2] = PR[90,2] + 16.425;
   1:L PR[91] R[100]mm/sec CNT100;
   1:  PR[91,1] = PR[90,1] + -18.799;
   1:  PR[91,2] = PR[90,2] + 17.763;
   1:L PR[91] R[100]mm/sec CNT100;
   1:  PR[91,1] = PR[90,1] + -23.072;
   1:  PR[91,2] = PR[90,2] + 18.170;
   1:L PR[91] R[100]mm/sec CNT100;
   1:  PR[91,1] = PR[90,1] + -27.313;
   1:  PR[91,2] = PR[90,2] + 17.630;
   1:L PR[91] R[100]mm/sec CNT100;
   1:  PR[91,1] = PR[90,1] + -31.320;
   1:  PR[91,2] = PR[90,2] + 16.182;
   1:L PR[91] R[100]mm/sec CNT100;
   1:  PR[91,1] = PR[90,1] + -32.483;
   1:  PR[91,2] = PR[90,2] + 15.448;
   1:L PR[91] R[100]mm/sec CNT100;
   1:  PR[91,1] = PR[90,1] + -34.882;
   1:  PR[91,2] = PR[90,2] + 13.908;
   1:L PR[91] R[100]mm/sec CNT100;
   1:  PR[91,1] = PR[90,1] + -37.851;
   1:  PR[91,2] = PR[90,2] + 10.916;
   1:L PR[91] R[100]mm/sec CNT100;
   1:  PR[91,1] = PR[90,1] + -40.075;
   1:  PR[91,2] = PR[90,2] + 7.361;
   1:L PR[91] R[100]mm/sec CNT100;
   1:  PR[91,1] = PR[90,1] + -41.451;
   1:  PR[91,2] = PR[90,2] + 3.415;
   1:L PR[91] R[100]mm/sec CNT100;
   1:  PR[91,1] = PR[90,1] + -41.677;
   1:  PR[91,2] = PR[90,2] + 1.423;
   1:L PR[91] R[100]mm/sec CNT100;
   1:  PR[91,1] = PR[90,1] + -41.728;
   1:  PR[91,2] = PR[90,2] + 1.173;
   1:L PR[91] R[100]mm/sec CNT100;
   1:  PR[91,1] = PR[90,1] + -41.940;
   1:  PR[91,2] = PR[90,2] + -0.717;
   1:L PR[91] R[100]mm/sec CNT100;
   1:  PR[91,1] = PR[90,1] + -41.702;
   1:  PR[91,2] = PR[90,2] + -2.633;
   1:L PR[91] R[100]mm/sec CNT100;
   1:  PR[91,1] = PR[90,1] + -41.451;
   1:  PR[91,2] = PR[90,2] + -4.875;
   1:L PR[91] R[100]mm/sec CNT100;
   1:  PR[91,1] = PR[90,1] + -40.075;
   1:  PR[91,2] = PR[90,2] + -8.820;
   1:L PR[91] R[100]mm/sec CNT100;
   1:  PR[91,1] = PR[90,1] + -37.851;
   1:  PR[91,2] = PR[90,2] + -12.375;
   1:L PR[91] R[100]mm/sec CNT100;
   1:  PR[91,1] = PR[90,1] + -34.884;
   1:  PR[91,2] = PR[90,2] + -15.365;
   1:L PR[91] R[100]mm/sec CNT100;
   1:  PR[91,1] = PR[90,1] + -31.315;
   1:  PR[91,2] = PR[90,2] + -17.643;
   1:L PR[91] R[100]mm/sec CNT100;
   1:  PR[91,1] = PR[90,1] + -27.313;
   1:  PR[91,2] = PR[90,2] + -19.089;
   1:L PR[91] R[100]mm/sec CNT100;
   1:  PR[91,1] = PR[90,1] + -23.072;
   1:  PR[91,2] = PR[90,2] + -19.629;
   1:L PR[91] R[100]mm/sec CNT100;
   1:  PR[91,1] = PR[90,1] + -18.799;
   1:  PR[91,2] = PR[90,2] + -19.222;
   1:L PR[91] R[100]mm/sec CNT100;
   1:  PR[91,1] = PR[90,1] + -14.709;
   1:  PR[91,2] = PR[90,2] + -17.884;
   1:L PR[91] R[100]mm/sec CNT100;
   1:  PR[91,1] = PR[90,1] + -10.999;
   1:  PR[91,2] = PR[90,2] + -15.659;
   1:L PR[91] R[100]mm/sec CNT100;
   1:  PR[91,1] = PR[90,1] + -7.803;
   1:  PR[91,2] = PR[90,2] + -12.683;
   1:L PR[91] R[100]mm/sec CNT100;
   1:  PR[91,1] = PR[90,1] + -7.750;
   1:  PR[91,2] = PR[90,2] + -12.614;
   1:L PR[91] R[100]mm/sec CNT100;
   1:  PR[91,1] = PR[90,1] + -5.412;
   1:  PR[91,2] = PR[90,2] + -9.139;
   1:L PR[91] R[100]mm/sec CNT100;
   1:  PR[91,1] = PR[90,1] + -5.269;
   1:  PR[91,2] = PR[90,2] + -8.824;
   1:L PR[91] R[100]mm/sec CNT100;
   1:  PR[91,1] = PR[90,1] + -3.898;
   1:  PR[91,2] = PR[90,2] + -5.146;
   1:L PR[91] R[100]mm/sec CNT100;
   1:  PR[91,1] = PR[90,1] + -3.803;
   1:  PR[91,2] = PR[90,2] + -4.644;
   1:L PR[91] R[100]mm/sec CNT100;
   1:  PR[91,1] = PR[90,1] + -3.342;
   1:  PR[91,2] = PR[90,2] + -0.824;
   1:L PR[91] R[100]mm/sec CNT100;
   1:  PR[91,1] = PR[90,1] + -3.341;
   1:  PR[91,2] = PR[90,2] + -0.821;
   1:L PR[91] R[100]mm/sec CNT100;
   1:  PR[91,1] = PR[90,1] + -3.814;
   1:  PR[91,2] = PR[90,2] + 3.101;
   1:L PR[91] R[100]mm/sec CNT100;
   1:  PR[91,1] = PR[90,1] + -3.819;
   1:  PR[91,2] = PR[90,2] + 3.270;
   1:L PR[91] R[100]mm/sec CNT100;
   1:  PR[91,1] = PR[90,1] + -3.897;
   1:  PR[91,2] = PR[90,2] + 3.686;
   1:L PR[91] R[100]mm/sec CNT100;
   1:  PR[91,1] = PR[90,1] + -5.269;
   1:  PR[91,2] = PR[90,2] + 7.364;
   1:L PR[91] R[100]mm/sec CNT100TB   .50sec,CALL END_PUD;
   1:  PR[92] = PR[91];
   1:  PR[92,3] = PR[92,3] + 20;
   1:J PR[92] 10% FINE;
   1:  PR[91,1] = PR[90,1] + -65.835;
   1:  PR[91,2] = PR[90,2] + 17.309;
   1:  PR[92] = PR[91];
   1:  PR[92,3] = PR[92,3] + 20;
   1:J PR[92] 10% FINE;
   1:L PR[91] R[100]mm/sec CNT100;
   1:  CALL LASER_DRAHT_START;
   1:  PR[91,1] = PR[90,1] + -67.251;
   1:  PR[91,2] = PR[90,2] + 17.568;
   1:L PR[91] R[100]mm/sec CNT100;
   1:  PR[91,1] = PR[90,1] + -69.905;
   1:  PR[91,2] = PR[90,2] + 18.028;
   1:L PR[91] R[100]mm/sec CNT100;
   1:  PR[91,1] = PR[90,1] + -72.104;
   1:  PR[91,2] = PR[90,2] + 17.985;
   1:L PR[91] R[100]mm/sec CNT100;
   1:  PR[91,1] = PR[90,1] + -74.021;
   1:  PR[91,2] = PR[90,2] + 17.930;
   1:L PR[91] R[100]mm/sec CNT100;
   1:  PR[91,1] = PR[90,1] + -76.804;
   1:  PR[91,2] = PR[90,2] + 17.308;
   1:L PR[91] R[100]mm/sec CNT100;
   1:  PR[91,1] = PR[90,1] + -78.006;
   1:  PR[91,2] = PR[90,2] + 17.028;
   1:L PR[91] R[100]mm/sec CNT100;
   1:  PR[91,1] = PR[90,1] + -81.701;
   1:  PR[91,2] = PR[90,2] + 15.366;
   1:L PR[91] R[100]mm/sec CNT100;
   1:  PR[91,1] = PR[90,1] + -84.943;
   1:  PR[91,2] = PR[90,2] + 13.028;
   1:L PR[91] R[100]mm/sec CNT100;
   1:  PR[91,1] = PR[90,1] + -87.601;
   1:  PR[91,2] = PR[90,2] + 10.120;
   1:L PR[91] R[100]mm/sec CNT100;
   1:  PR[91,1] = PR[90,1] + -89.553;
   1:  PR[91,2] = PR[90,2] + 6.770;
   1:L PR[91] R[100]mm/sec CNT100;
   1:  PR[91,1] = PR[90,1] + -90.754;
   1:  PR[91,2] = PR[90,2] + 3.074;
   1:L PR[91] R[100]mm/sec CNT100;
   1:  PR[91,1] = PR[90,1] + -90.794;
   1:  PR[91,2] = PR[90,2] + 2.786;
   1:L PR[91] R[100]mm/sec CNT100;
   1:  PR[91,1] = PR[90,1] + -91.160;
   1:  PR[91,2] = PR[90,2] + -0.669;
   1:L PR[91] R[100]mm/sec CNT100;
   1:  PR[91,1] = PR[90,1] + -90.974;
   1:  PR[91,2] = PR[90,2] + -1.462;
   1:L PR[91] R[100]mm/sec CNT100;
   1:  PR[91,1] = PR[90,1] + -90.649;
   1:  PR[91,2] = PR[90,2] + -4.563;
   1:L PR[91] R[100]mm/sec CNT100;
   1:  PR[91,1] = PR[90,1] + -90.399;
   1:  PR[91,2] = PR[90,2] + -5.327;
   1:L PR[91] R[100]mm/sec CNT100;
   1:  PR[91,1] = PR[90,1] + -89.453;
   1:  PR[91,2] = PR[90,2] + -8.240;
   1:L PR[91] R[100]mm/sec CNT100;
   1:  PR[91,1] = PR[90,1] + -87.510;
   1:  PR[91,2] = PR[90,2] + -11.599;
   1:L PR[91] R[100]mm/sec CNT100;
   1:  PR[91,1] = PR[90,1] + -84.901;
   1:  PR[91,2] = PR[90,2] + -14.503;
   1:L PR[91] R[100]mm/sec CNT100;
   1:  PR[91,1] = PR[90,1] + -81.734;
   1:  PR[91,2] = PR[90,2] + -16.822;
   1:L PR[91] R[100]mm/sec CNT100;
   1:  PR[91,1] = PR[90,1] + -78.088;
   1:  PR[91,2] = PR[90,2] + -18.470;
   1:L PR[91] R[100]mm/sec CNT100;
   1:  PR[91,1] = PR[90,1] + -74.068;
   1:  PR[91,2] = PR[90,2] + -19.378;
   1:L PR[91] R[100]mm/sec CNT100;
   1:  PR[91,1] = PR[90,1] + -70.781;
   1:  PR[91,2] = PR[90,2] + -19.450;
   1:L PR[91] R[100]mm/sec CNT100;
   1:  PR[91,1] = PR[90,1] + -69.897;
   1:  PR[91,2] = PR[90,2] + -19.483;
   1:L PR[91] R[100]mm/sec CNT100;
   1:  PR[91,1] = PR[90,1] + -67.185;
   1:  PR[91,2] = PR[90,2] + -18.997;
   1:L PR[91] R[100]mm/sec CNT100;
   1:  PR[91,1] = PR[90,1] + -65.779;
   1:  PR[91,2] = PR[90,2] + -18.768;
   1:L PR[91] R[100]mm/sec CNT100;
   1:  PR[91,1] = PR[90,1] + -63.752;
   1:  PR[91,2] = PR[90,2] + -17.961;
   1:L PR[91] R[100]mm/sec CNT100;
   1:  PR[91,1] = PR[90,1] + -61.885;
   1:  PR[91,2] = PR[90,2] + -17.252;
   1:L PR[91] R[100]mm/sec CNT100;
   1:  PR[91,1] = PR[90,1] + -60.564;
   1:  PR[91,2] = PR[90,2] + -16.379;
   1:L PR[91] R[100]mm/sec CNT100;
   1:  PR[91,1] = PR[90,1] + -58.389;
   1:  PR[91,2] = PR[90,2] + -14.988;
   1:L PR[91] R[100]mm/sec CNT100;
   1:  PR[91,1] = PR[90,1] + -57.698;
   1:  PR[91,2] = PR[90,2] + -14.284;
   1:L PR[91] R[100]mm/sec CNT100;
   1:  PR[91,1] = PR[90,1] + -55.455;
   1:  PR[91,2] = PR[90,2] + -12.058;
   1:L PR[91] R[100]mm/sec CNT100;
   1:  PR[91,1] = PR[90,1] + -53.244;
   1:  PR[91,2] = PR[90,2] + -8.601;
   1:L PR[91] R[100]mm/sec CNT100;
   1:  PR[91,1] = PR[90,1] + -52.306;
   1:  PR[91,2] = PR[90,2] + -5.987;
   1:L PR[91] R[100]mm/sec CNT100;
   1:  PR[91,1] = PR[90,1] + -51.827;
   1:  PR[91,2] = PR[90,2] + -4.736;
   1:L PR[91] R[100]mm/sec CNT100;
   1:  PR[91,1] = PR[90,1] + -51.339;
   1:  PR[91,2] = PR[90,2] + -0.808;
   1:L PR[91] R[100]mm/sec CNT100;
   1:  PR[91,1] = PR[90,1] + -51.335;
   1:  PR[91,2] = PR[90,2] + -0.743;
   1:L PR[91] R[100]mm/sec CNT100;
   1:  PR[91,1] = PR[90,1] + -51.543;
   1:  PR[91,2] = PR[90,2] + 1.740;
   1:L PR[91] R[100]mm/sec CNT100;
   1:  PR[91,1] = PR[90,1] + -51.729;
   1:  PR[91,2] = PR[90,2] + 3.294;
   1:L PR[91] R[100]mm/sec CNT100;
   1:  PR[91,1] = PR[90,1] + -53.158;
   1:  PR[91,2] = PR[90,2] + 7.120;
   1:L PR[91] R[100]mm/sec CNT100;
   1:  PR[91,1] = PR[90,1] + -55.454;
   1:  PR[91,2] = PR[90,2] + 10.569;
   1:L PR[91] R[100]mm/sec CNT100;
   1:  PR[91,1] = PR[90,1] + -58.503;
   1:  PR[91,2] = PR[90,2] + 13.501;
   1:L PR[91] R[100]mm/sec CNT100;
   1:  PR[91,1] = PR[90,1] + -61.978;
   1:  PR[91,2] = PR[90,2] + 15.784;
   1:L PR[91] R[100]mm/sec CNT100;
   1:  PR[91,1] = PR[90,1] + -65.835;
   1:  PR[91,2] = PR[90,2] + 17.309;
   1:L PR[91] R[100]mm/sec CNT100TB   .50sec,CALL END_PUD;
   1:  PR[92] = PR[91];
   1:  PR[92,3] = PR[92,3] + 20;
   1:J PR[92] 10% FINE;
   1:  PR[91] = PR[90];
   1:  PR[91,1] = PR[90,1] + 54.067;
   1:  PR[91,2] = PR[90,2] + -13.931;
   1:  PR[91,3] = PR[90,3] + 31.395;
   1:  PR[92] = PR[91];
   1:  PR[92,3] = PR[92,3] + 20;
   1:J PR[92] 10% FINE;
   1:L PR[91] R[100]mm/sec CNT100;
   1:  CALL LASER_DRAHT_START;
   1:  PR[91,1] = PR[90,1] + 56.524;
   1:  PR[91,2] = PR[90,2] + -15.899;
   1:L PR[91] R[100]mm/sec CNT100;
   1:  PR[91,1] = PR[90,1] + 57.775;
   1:  PR[91,2] = PR[90,2] + -16.769;
   1:L PR[91] R[100]mm/sec CNT100;
   1:  PR[91,1] = PR[90,1] + 61.953;
   1:  PR[91,2] = PR[90,2] + -18.788;
   1:L PR[91] R[100]mm/sec CNT100;
   1:  PR[91,1] = PR[90,1] + 66.520;
   1:  PR[91,2] = PR[90,2] + -20.043;
   1:L PR[91] R[100]mm/sec CNT100;
   1:  PR[91,1] = PR[90,1] + 67.435;
   1:  PR[91,2] = PR[90,2] + -20.108;
   1:L PR[91] R[100]mm/sec CNT100;
   1:  PR[91,1] = PR[90,1] + 71.167;
   1:  PR[91,2] = PR[90,2] + -20.319;
   1:L PR[91] R[100]mm/sec CNT100;
   1:  PR[91,1] = PR[90,1] + 73.113;
   1:  PR[91,2] = PR[90,2] + -20.042;
   1:L PR[91] R[100]mm/sec CNT100;
   1:  PR[91,1] = PR[90,1] + 75.714;
   1:  PR[91,2] = PR[90,2] + -19.634;
   1:L PR[91] R[100]mm/sec CNT100;
   1:  PR[91,1] = PR[90,1] + 78.353;
   1:  PR[91,2] = PR[90,2] + -18.661;
   1:L PR[91] R[100]mm/sec CNT100;
   1:  PR[91,1] = PR[90,1] + 79.955;
   1:  PR[91,2] = PR[90,2] + -18.047;
   1:L PR[91] R[100]mm/sec CNT100;
   1:  PR[91,1] = PR[90,1] + 82.863;
   1:  PR[91,2] = PR[90,2] + -16.194;
   1:L PR[91] R[100]mm/sec CNT100;
   1:  PR[91,1] = PR[90,1] + 83.702;
   1:  PR[91,2] = PR[90,2] + -15.646;
   1:L PR[91] R[100]mm/sec CNT100;
   1:  PR[91,1] = PR[90,1] + 86.454;
   1:  PR[91,2] = PR[90,2] + -12.900;
   1:L PR[91] R[100]mm/sec CNT100;
   1:  PR[91,1] = PR[90,1] + 86.793;
   1:  PR[91,2] = PR[90,2] + -12.555;
   1:L PR[91] R[100]mm/sec CNT100;
   1:  PR[91,1] = PR[90,1] + 89.100;
   1:  PR[91,2] = PR[90,2] + -8.917;
   1:L PR[91] R[100]mm/sec CNT100;
   1:  PR[91,1] = PR[90,1] + 90.519;
   1:  PR[91,2] = PR[90,2] + -4.915;
   1:L PR[91] R[100]mm/sec CNT100;
   1:  PR[91,1] = PR[90,1] + 91.005;
   1:  PR[91,2] = PR[90,2] + -0.729;
   1:L PR[91] R[100]mm/sec CNT100;
   1:  PR[91,1] = PR[90,1] + 90.519;
   1:  PR[91,2] = PR[90,2] + 3.456;
   1:L PR[91] R[100]mm/sec CNT100;
   1:  PR[91,1] = PR[90,1] + 89.100;
   1:  PR[91,2] = PR[90,2] + 7.458;
   1:L PR[91] R[100]mm/sec CNT100;
   1:  PR[91,1] = PR[90,1] + 86.797;
   1:  PR[91,2] = PR[90,2] + 11.089;
   1:L PR[91] R[100]mm/sec CNT100;
   1:  PR[91,1] = PR[90,1] + 83.710;
   1:  PR[91,2] = PR[90,2] + 14.178;
   1:L PR[91] R[100]mm/sec CNT100;
   1:  PR[91,1] = PR[90,1] + 80.939;
   1:  PR[91,2] = PR[90,2] + 15.939;
   1:L PR[91] R[100]mm/sec CNT100;
   1:  PR[91,1] = PR[90,1] + 79.955;
   1:  PR[91,2] = PR[90,2] + 16.585;
   1:L PR[91] R[100]mm/sec CNT100;
   1:  PR[91,1] = PR[90,1] + 77.344;
   1:  PR[91,2] = PR[90,2] + 17.541;
   1:L PR[91] R[100]mm/sec CNT100;
   1:  PR[91,1] = PR[90,1] + 75.714;
   1:  PR[91,2] = PR[90,2] + 18.171;
   1:L PR[91] R[100]mm/sec CNT100;
   1:  PR[91,1] = PR[90,1] + 73.559;
   1:  PR[91,2] = PR[90,2] + 18.473;
   1:L PR[91] R[100]mm/sec CNT100;
   1:  PR[91,1] = PR[90,1] + 71.167;
   1:  PR[91,2] = PR[90,2] + 18.856;
   1:L PR[91] R[100]mm/sec CNT100;
   1:  PR[91,1] = PR[90,1] + 69.715;
   1:  PR[91,2] = PR[90,2] + 18.748;
   1:L PR[91] R[100]mm/sec CNT100;
   1:  PR[91,1] = PR[90,1] + 66.521;
   1:  PR[91,2] = PR[90,2] + 18.580;
   1:L PR[91] R[100]mm/sec CNT100;
   1:  PR[91,1] = PR[90,1] + 65.913;
   1:  PR[91,2] = PR[90,2] + 18.400;
   1:L PR[91] R[100]mm/sec CNT100;
   1:  PR[91,1] = PR[90,1] + 61.871;
   1:  PR[91,2] = PR[90,2] + 17.296;
   1:L PR[91] R[100]mm/sec CNT100;
   1:  PR[91,1] = PR[90,1] + 57.776;
   1:  PR[91,2] = PR[90,2] + 15.311;
   1:L PR[91] R[100]mm/sec CNT100;
   1:  PR[91,1] = PR[90,1] + 56.524;
   1:  PR[91,2] = PR[90,2] + 14.440;
   1:L PR[91] R[100]mm/sec CNT100;
   1:  PR[91,1] = PR[90,1] + 54.067;
   1:  PR[91,2] = PR[90,2] + 12.472;
   1:L PR[91] R[100]mm/sec CNT100;
   1:  PR[91,1] = PR[90,1] + 52.041;
   1:  PR[91,2] = PR[90,2] + 10.120;
   1:L PR[91] R[100]mm/sec CNT100;
   1:  PR[91,1] = PR[90,1] + 50.998;
   1:  PR[91,2] = PR[90,2] + 8.764;
   1:L PR[91] R[100]mm/sec CNT100;
   1:  PR[91,1] = PR[90,1] + 49.187;
   1:  PR[91,2] = PR[90,2] + 4.915;
   1:L PR[91] R[100]mm/sec CNT100;
   1:  PR[91,1] = PR[90,1] + 48.923;
   1:  PR[91,2] = PR[90,2] + 4.292;
   1:L PR[91] R[100]mm/sec CNT100;
   1:  PR[91,1] = PR[90,1] + 48.166;
   1:  PR[91,2] = PR[90,2] + -0.709;
   1:L PR[91] R[100]mm/sec CNT100;
   1:  PR[91,1] = PR[90,1] + 48.210;
   1:  PR[91,2] = PR[90,2] + -1.088;
   1:L PR[91] R[100]mm/sec CNT100;
   1:  PR[91,1] = PR[90,1] + 48.922;
   1:  PR[91,2] = PR[90,2] + -5.748;
   1:L PR[91] R[100]mm/sec CNT100;
   1:  PR[91,1] = PR[90,1] + 49.186;
   1:  PR[91,2] = PR[90,2] + -6.372;
   1:L PR[91] R[100]mm/sec CNT100;
   1:  PR[91,1] = PR[90,1] + 50.997;
   1:  PR[91,2] = PR[90,2] + -10.222;
   1:L PR[91] R[100]mm/sec CNT100;
   1:  PR[91,1] = PR[90,1] + 52.041;
   1:  PR[91,2] = PR[90,2] + -11.578;
   1:L PR[91] R[100]mm/sec CNT100;
   1:  PR[91,1] = PR[90,1] + 54.067;
   1:  PR[91,2] = PR[90,2] + -13.931;
   1:L PR[91] R[100]mm/sec CNT100TB   .50sec,CALL END_PUD;
   1:  PR[92] = PR[91];
   1:  PR[92,3] = PR[92,3] + 20;
   1:J PR[92] 10% FINE;
   1:  PR[91,1] = PR[90,1] + 41.310;
   1:  PR[91,2] = PR[90,2] + 8.698;
   1:  PR[92] = PR[91];
   1:  PR[92,3] = PR[92,3] + 20;
   1:J PR[92] 10% FINE;
   1:L PR[91] R[100]mm/sec CNT100;
   1:  CALL LASER_DRAHT_START;
   1:  PR[91,1] = PR[90,1] + 41.139;
   1:  PR[91,2] = PR[90,2] + 9.014;
   1:L PR[91] R[100]mm/sec CNT100;
   1:  PR[91,1] = PR[90,1] + 39.627;
   1:  PR[91,2] = PR[90,2] + 11.001;
   1:L PR[91] R[100]mm/sec CNT100;
   1:  PR[91,1] = PR[90,1] + 37.965;
   1:  PR[91,2] = PR[90,2] + 13.114;
   1:L PR[91] R[100]mm/sec CNT100;
   1:  PR[91,1] = PR[90,1] + 36.139;
   1:  PR[91,2] = PR[90,2] + 14.523;
   1:L PR[91] R[100]mm/sec CNT100;
   1:  PR[91,1] = PR[90,1] + 33.939;
   1:  PR[91,2] = PR[90,2] + 16.180;
   1:L PR[91] R[100]mm/sec CNT100;
   1:  PR[91,1] = PR[90,1] + 31.882;
   1:  PR[91,2] = PR[90,2] + 17.040;
   1:L PR[91] R[100]mm/sec CNT100;
   1:  PR[91,1] = PR[90,1] + 29.256;
   1:  PR[91,2] = PR[90,2] + 18.110;
   1:L PR[91] R[100]mm/sec CNT100;
   1:  PR[91,1] = PR[90,1] + 24.218;
   1:  PR[91,2] = PR[90,2] + 18.774;
   1:L PR[91] R[100]mm/sec CNT100;
   1:  PR[91,1] = PR[90,1] + 19.174;
   1:  PR[91,2] = PR[90,2] + 18.114;
   1:L PR[91] R[100]mm/sec CNT100;
   1:  PR[91,1] = PR[90,1] + 17.373;
   1:  PR[91,2] = PR[90,2] + 17.377;
   1:L PR[91] R[100]mm/sec CNT100;
   1:  PR[91,1] = PR[90,1] + 14.470;
   1:  PR[91,2] = PR[90,2] + 16.176;
   1:L PR[91] R[100]mm/sec CNT100;
   1:  PR[91,1] = PR[90,1] + 10.419;
   1:  PR[91,2] = PR[90,2] + 13.082;
   1:L PR[91] R[100]mm/sec CNT100;
   1:  PR[91,1] = PR[90,1] + 7.306;
   1:  PR[91,2] = PR[90,2] + 9.041;
   1:L PR[91] R[100]mm/sec CNT100;
   1:  PR[91,1] = PR[90,1] + 6.644;
   1:  PR[91,2] = PR[90,2] + 7.450;
   1:L PR[91] R[100]mm/sec CNT100;
   1:  PR[91,1] = PR[90,1] + 5.348;
   1:  PR[91,2] = PR[90,2] + 4.331;
   1:L PR[91] R[100]mm/sec CNT100;
   1:  PR[91,1] = PR[90,1] + 4.679;
   1:  PR[91,2] = PR[90,2] + -0.729;
   1:L PR[91] R[100]mm/sec CNT100;
   1:  PR[91,1] = PR[90,1] + 5.349;
   1:  PR[91,2] = PR[90,2] + -5.793;
   1:L PR[91] R[100]mm/sec CNT100;
   1:  PR[91,1] = PR[90,1] + 7.310;
   1:  PR[91,2] = PR[90,2] + -10.507;
   1:L PR[91] R[100]mm/sec CNT100;
   1:  PR[91,1] = PR[90,1] + 9.337;
   1:  PR[91,2] = PR[90,2] + -13.137;
   1:L PR[91] R[100]mm/sec CNT100;
   1:  PR[91,1] = PR[90,1] + 10.425;
   1:  PR[91,2] = PR[90,2] + -14.548;
   1:L PR[91] R[100]mm/sec CNT100;
   1:  PR[91,1] = PR[90,1] + 14.481;
   1:  PR[91,2] = PR[90,2] + -17.640;
   1:L PR[91] R[100]mm/sec CNT100;
   1:  PR[91,1] = PR[90,1] + 19.193;
   1:  PR[91,2] = PR[90,2] + -19.578;
   1:L PR[91] R[100]mm/sec CNT100;
   1:  PR[91,1] = PR[90,1] + 22.207;
   1:  PR[91,2] = PR[90,2] + -19.974;
   1:L PR[91] R[100]mm/sec CNT100;
   1:  PR[91,1] = PR[90,1] + 24.235;
   1:  PR[91,2] = PR[90,2] + -20.233;
   1:L PR[91] R[100]mm/sec CNT100;
   1:  PR[91,1] = PR[90,1] + 29.272;
   1:  PR[91,2] = PR[90,2] + -19.564;
   1:L PR[91] R[100]mm/sec CNT100;
   1:  PR[91,1] = PR[90,1] + 33.962;
   1:  PR[91,2] = PR[90,2] + -17.625;
   1:L PR[91] R[100]mm/sec CNT100;
   1:  PR[91,1] = PR[90,1] + 36.158;
   1:  PR[91,2] = PR[90,2] + -15.963;
   1:L PR[91] R[100]mm/sec CNT100;
   1:  PR[91,1] = PR[90,1] + 37.983;
   1:  PR[91,2] = PR[90,2] + -14.556;
   1:L PR[91] R[100]mm/sec CNT100;
   1:  PR[91,1] = PR[90,1] + 39.652;
   1:  PR[91,2] = PR[90,2] + -12.419;
   1:L PR[91] R[100]mm/sec CNT100;
   1:  PR[91,1] = PR[90,1] + 41.138;
   1:  PR[91,2] = PR[90,2] + -10.475;
   1:L PR[91] R[100]mm/sec CNT100;
   1:  PR[91,1] = PR[90,1] + 41.275;
   1:  PR[91,2] = PR[90,2] + -10.225;
   1:L PR[91] R[100]mm/sec CNT100;
   1:  PR[91,1] = PR[90,1] + 42.172;
   1:  PR[91,2] = PR[90,2] + -8.051;
   1:L PR[91] R[100]mm/sec CNT100;
   1:  PR[91,1] = PR[90,1] + 42.758;
   1:  PR[91,2] = PR[90,2] + -6.742;
   1:L PR[91] R[100]mm/sec CNT100;
   1:  PR[91,1] = PR[90,1] + 43.359;
   1:  PR[91,2] = PR[90,2] + -4.389;
   1:L PR[91] R[100]mm/sec CNT100;
   1:  PR[91,1] = PR[90,1] + 43.445;
   1:  PR[91,2] = PR[90,2] + -3.736;
   1:L PR[91] R[100]mm/sec CNT100;
   1:  PR[91,1] = PR[90,1] + 43.707;
   1:  PR[91,2] = PR[90,2] + -0.772;
   1:L PR[91] R[100]mm/sec CNT100;
   1:  PR[91,1] = PR[90,1] + 43.683;
   1:  PR[91,2] = PR[90,2] + -0.589;
   1:L PR[91] R[100]mm/sec CNT100;
   1:  PR[91,1] = PR[90,1] + 43.369;
   1:  PR[91,2] = PR[90,2] + 2.862;
   1:L PR[91] R[100]mm/sec CNT100;
   1:  PR[91,1] = PR[90,1] + 42.695;
   1:  PR[91,2] = PR[90,2] + 5.468;
   1:L PR[91] R[100]mm/sec CNT100;
   1:  PR[91,1] = PR[90,1] + 42.093;
   1:  PR[91,2] = PR[90,2] + 6.927;
   1:L PR[91] R[100]mm/sec CNT100;
   1:  PR[91,1] = PR[90,1] + 41.310;
   1:  PR[91,2] = PR[90,2] + 8.698;
   1:L PR[91] R[100]mm/sec CNT100TB   .50sec,CALL END_PUD;
   1:  PR[92] = PR[91];
   1:  PR[92,3] = PR[92,3] + 20;
   1:J PR[92] 10% FINE;
   1:  PR[91,1] = PR[90,1] + -6.984;
   1:  PR[91,2] = PR[90,2] + -12.298;
   1:  PR[92] = PR[91];
   1:  PR[92,3] = PR[92,3] + 20;
   1:J PR[92] 10% FINE;
   1:L PR[91] R[100]mm/sec CNT100;
   1:  CALL LASER_DRAHT_START;
   1:  PR[91,1] = PR[90,1] + -5.016;
   1:  PR[91,2] = PR[90,2] + -9.371;
   1:L PR[91] R[100]mm/sec CNT100;
   1:  PR[91,1] = PR[90,1] + -4.586;
   1:  PR[91,2] = PR[90,2] + -8.422;
   1:L PR[91] R[100]mm/sec CNT100;
   1:  PR[91,1] = PR[90,1] + -3.447;
   1:  PR[91,2] = PR[90,2] + -5.368;
   1:L PR[91] R[100]mm/sec CNT100;
   1:  PR[91,1] = PR[90,1] + -3.223;
   1:  PR[91,2] = PR[90,2] + -4.180;
   1:L PR[91] R[100]mm/sec CNT100;
   1:  PR[91,1] = PR[90,1] + -2.843;
   1:  PR[91,2] = PR[90,2] + -1.030;
   1:L PR[91] R[100]mm/sec CNT100;
   1:  PR[91,1] = PR[90,1] + -2.837;
   1:  PR[91,2] = PR[90,2] + -0.821;
   1:L PR[91] R[100]mm/sec CNT100;
   1:  PR[91,1] = PR[90,1] + -3.226;
   1:  PR[91,2] = PR[90,2] + 2.415;
   1:L PR[91] R[100]mm/sec CNT100;
   1:  PR[91,1] = PR[90,1] + -3.239;
   1:  PR[91,2] = PR[90,2] + 2.803;
   1:L PR[91] R[100]mm/sec CNT100;
   1:  PR[91,1] = PR[90,1] + -3.445;
   1:  PR[91,2] = PR[90,2] + 3.905;
   1:L PR[91] R[100]mm/sec CNT100;
   1:  PR[91,1] = PR[90,1] + -4.585;
   1:  PR[91,2] = PR[90,2] + 6.960;
   1:L PR[91] R[100]mm/sec CNT100;
   1:  PR[91,1] = PR[90,1] + -5.014;
   1:  PR[91,2] = PR[90,2] + 7.909;
   1:L PR[91] R[100]mm/sec CNT100;
   1:  PR[91,1] = PR[90,1] + -6.983;
   1:  PR[91,2] = PR[90,2] + 10.836;
   1:L PR[91] R[100]mm/sec CNT100;
   1:  PR[91,1] = PR[90,1] + -7.457;
   1:  PR[91,2] = PR[90,2] + 11.450;
   1:L PR[91] R[100]mm/sec CNT100;
   1:  PR[91,1] = PR[90,1] + -10.305;
   1:  PR[91,2] = PR[90,2] + 14.095;
   1:L PR[91] R[100]mm/sec CNT100;
   1:  PR[91,1] = PR[90,1] + -10.633;
   1:  PR[91,2] = PR[90,2] + 14.361;
   1:L PR[91] R[100]mm/sec CNT100;
   1:  PR[91,1] = PR[90,1] + -14.364;
   1:  PR[91,2] = PR[90,2] + 16.511;
   1:L PR[91] R[100]mm/sec CNT100;
   1:  PR[91,1] = PR[90,1] + -14.377;
   1:  PR[91,2] = PR[90,2] + 16.517;
   1:L PR[91] R[100]mm/sec CNT100;
   1:  PR[91,1] = PR[90,1] + -16.694;
   1:  PR[91,2] = PR[90,2] + 17.235;
   1:L PR[91] R[100]mm/sec CNT100;
   1:  PR[91,1] = PR[90,1] + -18.585;
   1:  PR[91,2] = PR[90,2] + 17.853;
   1:L PR[91] R[100]mm/sec CNT100;
   1:  PR[91,1] = PR[90,1] + -22.887;
   1:  PR[91,2] = PR[90,2] + 18.257;
   1:L PR[91] R[100]mm/sec CNT100;
   1:  PR[91,1] = PR[90,1] + -23.181;
   1:  PR[91,2] = PR[90,2] + 18.222;
   1:L PR[91] R[100]mm/sec CNT100;
   1:  PR[91,1] = PR[90,1] + -27.137;
   1:  PR[91,2] = PR[90,2] + 17.710;
   1:L PR[91] R[100]mm/sec CNT100;
   1:  PR[91,1] = PR[90,1] + -31.156;
   1:  PR[91,2] = PR[90,2] + 16.254;
   1:L PR[91] R[100]mm/sec CNT100;
   1:  PR[91,1] = PR[90,1] + -34.738;
   1:  PR[91,2] = PR[90,2] + 13.964;
   1:L PR[91] R[100]mm/sec CNT100;
   1:  PR[91,1] = PR[90,1] + -37.714;
   1:  PR[91,2] = PR[90,2] + 10.961;
   1:L PR[91] R[100]mm/sec CNT100;
   1:  PR[91,1] = PR[90,1] + -39.945;
   1:  PR[91,2] = PR[90,2] + 7.391;
   1:L PR[91] R[100]mm/sec CNT100;
   1:  PR[91,1] = PR[90,1] + -41.325;
   1:  PR[91,2] = PR[90,2] + 3.430;
   1:L PR[91] R[100]mm/sec CNT100;
   1:  PR[91,1] = PR[90,1] + -41.504;
   1:  PR[91,2] = PR[90,2] + 1.857;
   1:L PR[91] R[100]mm/sec CNT100;
   1:  PR[91,1] = PR[90,1] + -41.545;
   1:  PR[91,2] = PR[90,2] + 1.656;
   1:L PR[91] R[100]mm/sec CNT100;
   1:  PR[91,1] = PR[90,1] + -41.811;
   1:  PR[91,2] = PR[90,2] + -0.717;
   1:L PR[91] R[100]mm/sec CNT100;
   1:  PR[91,1] = PR[90,1] + -41.624;
   1:  PR[91,2] = PR[90,2] + -2.220;
   1:L PR[91] R[100]mm/sec CNT100;
   1:  PR[91,1] = PR[90,1] + -41.325;
   1:  PR[91,2] = PR[90,2] + -4.890;
   1:L PR[91] R[100]mm/sec CNT100;
   1:  PR[91,1] = PR[90,1] + -39.945;
   1:  PR[91,2] = PR[90,2] + -8.850;
   1:L PR[91] R[100]mm/sec CNT100;
   1:  PR[91,1] = PR[90,1] + -37.714;
   1:  PR[91,2] = PR[90,2] + -12.419;
   1:L PR[91] R[100]mm/sec CNT100;
   1:  PR[91,1] = PR[90,1] + -34.738;
   1:  PR[91,2] = PR[90,2] + -15.423;
   1:L PR[91] R[100]mm/sec CNT100;
   1:  PR[91,1] = PR[90,1] + -31.156;
   1:  PR[91,2] = PR[90,2] + -17.713;
   1:L PR[91] R[100]mm/sec CNT100;
   1:  PR[91,1] = PR[90,1] + -27.138;
   1:  PR[91,2] = PR[90,2] + -19.169;
   1:L PR[91] R[100]mm/sec CNT100;
   1:  PR[91,1] = PR[90,1] + -22.878;
   1:  PR[91,2] = PR[90,2] + -19.715;
   1:L PR[91] R[100]mm/sec CNT100;
   1:  PR[91,1] = PR[90,1] + -18.585;
   1:  PR[91,2] = PR[90,2] + -19.311;
   1:L PR[91] R[100]mm/sec CNT100;
   1:  PR[91,1] = PR[90,1] + -16.694;
   1:  PR[91,2] = PR[90,2] + -18.694;
   1:L PR[91] R[100]mm/sec CNT100;
   1:  PR[91,1] = PR[90,1] + -14.376;
   1:  PR[91,2] = PR[90,2] + -17.976;
   1:L PR[91] R[100]mm/sec CNT100;
   1:  PR[91,1] = PR[90,1] + -14.364;
   1:  PR[91,2] = PR[90,2] + -17.970;
   1:L PR[91] R[100]mm/sec CNT100;
   1:  PR[91,1] = PR[90,1] + -10.634;
   1:  PR[91,2] = PR[90,2] + -15.821;
   1:L PR[91] R[100]mm/sec CNT100;
   1:  PR[91,1] = PR[90,1] + -10.307;
   1:  PR[91,2] = PR[90,2] + -15.555;
   1:L PR[91] R[100]mm/sec CNT100;
   1:  PR[91,1] = PR[90,1] + -7.459;
   1:  PR[91,2] = PR[90,2] + -12.910;
   1:L PR[91] R[100]mm/sec CNT100;
   1:  PR[91,1] = PR[90,1] + -6.984;
   1:  PR[91,2] = PR[90,2] + -12.298;
   1:L PR[91] R[100]mm/sec CNT100TB   .50sec,CALL END_PUD;
   1:  PR[92] = PR[91];
   1:  PR[92,3] = PR[92,3] + 20;
   1:J PR[92] 10% FINE;
   1:  PR[91,1] = PR[90,1] + -50.624;
   1:  PR[91,2] = PR[90,2] + -1.776;
   1:  PR[92] = PR[91];
   1:  PR[92,3] = PR[92,3] + 20;
   1:J PR[92] 10% FINE;
   1:L PR[91] R[100]mm/sec CNT100;
   1:  CALL LASER_DRAHT_START;
   1:  PR[91,1] = PR[90,1] + -50.552;
   1:  PR[91,2] = PR[90,2] + -0.743;
   1:L PR[91] R[100]mm/sec CNT100;
   1:  PR[91,1] = PR[90,1] + -50.671;
   1:  PR[91,2] = PR[90,2] + 0.667;
   1:L PR[91] R[100]mm/sec CNT100;
   1:  PR[91,1] = PR[90,1] + -50.990;
   1:  PR[91,2] = PR[90,2] + 3.333;
   1:L PR[91] R[100]mm/sec CNT100;
   1:  PR[91,1] = PR[90,1] + -52.439;
   1:  PR[91,2] = PR[90,2] + 7.197;
   1:L PR[91] R[100]mm/sec CNT100;
   1:  PR[91,1] = PR[90,1] + -53.729;
   1:  PR[91,2] = PR[90,2] + 9.141;
   1:L PR[91] R[100]mm/sec CNT100;
   1:  PR[91,1] = PR[90,1] + -54.759;
   1:  PR[91,2] = PR[90,2] + 10.668;
   1:L PR[91] R[100]mm/sec CNT100;
   1:  PR[91,1] = PR[90,1] + -57.832;
   1:  PR[91,2] = PR[90,2] + 13.604;
   1:L PR[91] R[100]mm/sec CNT100;
   1:  PR[91,1] = PR[90,1] + -61.506;
   1:  PR[91,2] = PR[90,2] + 15.875;
   1:L PR[91] R[100]mm/sec CNT100;
   1:  PR[91,1] = PR[90,1] + -65.421;
   1:  PR[91,2] = PR[90,2] + 17.406;
   1:L PR[91] R[100]mm/sec CNT100;
   1:  PR[91,1] = PR[90,1] + -69.521;
   1:  PR[91,2] = PR[90,2] + 18.124;
   1:L PR[91] R[100]mm/sec CNT100;
   1:  PR[91,1] = PR[90,1] + -73.660;
   1:  PR[91,2] = PR[90,2] + 18.018;
   1:L PR[91] R[100]mm/sec CNT100;
   1:  PR[91,1] = PR[90,1] + -77.665;
   1:  PR[91,2] = PR[90,2] + 17.105;
   1:L PR[91] R[100]mm/sec CNT100;
   1:  PR[91,1] = PR[90,1] + -81.369;
   1:  PR[91,2] = PR[90,2] + 15.433;
   1:L PR[91] R[100]mm/sec CNT100;
   1:  PR[91,1] = PR[90,1] + -84.621;
   1:  PR[91,2] = PR[90,2] + 13.083;
   1:L PR[91] R[100]mm/sec CNT100;
   1:  PR[91,1] = PR[90,1] + -87.291;
   1:  PR[91,2] = PR[90,2] + 10.158;
   1:L PR[91] R[100]mm/sec CNT100;
   1:  PR[91,1] = PR[90,1] + -89.275;
   1:  PR[91,2] = PR[90,2] + 6.786;
   1:L PR[91] R[100]mm/sec CNT100;
   1:  PR[91,1] = PR[90,1] + -90.495;
   1:  PR[91,2] = PR[90,2] + 3.105;
   1:L PR[91] R[100]mm/sec CNT100;
   1:  PR[91,1] = PR[90,1] + -90.905;
   1:  PR[91,2] = PR[90,2] + -0.673;
   1:L PR[91] R[100]mm/sec CNT100;
   1:  PR[91,1] = PR[90,1] + -90.823;
   1:  PR[91,2] = PR[90,2] + -1.023;
   1:L PR[91] R[100]mm/sec CNT100;
   1:  PR[91,1] = PR[90,1] + -90.451;
   1:  PR[91,2] = PR[90,2] + -4.573;
   1:L PR[91] R[100]mm/sec CNT100;
   1:  PR[91,1] = PR[90,1] + -90.339;
   1:  PR[91,2] = PR[90,2] + -4.915;
   1:L PR[91] R[100]mm/sec CNT100;
   1:  PR[91,1] = PR[90,1] + -89.252;
   1:  PR[91,2] = PR[90,2] + -8.259;
   1:L PR[91] R[100]mm/sec CNT100;
   1:  PR[91,1] = PR[90,1] + -87.305;
   1:  PR[91,2] = PR[90,2] + -11.628;
   1:L PR[91] R[100]mm/sec CNT100;
   1:  PR[91,1] = PR[90,1] + -84.698;
   1:  PR[91,2] = PR[90,2] + -14.534;
   1:L PR[91] R[100]mm/sec CNT100;
   1:  PR[91,1] = PR[90,1] + -81.441;
   1:  PR[91,2] = PR[90,2] + -16.878;
   1:L PR[91] R[100]mm/sec CNT100;
   1:  PR[91,1] = PR[90,1] + -77.708;
   1:  PR[91,2] = PR[90,2] + -18.554;
   1:L PR[91] R[100]mm/sec CNT100;
   1:  PR[91,1] = PR[90,1] + -74.560;
   1:  PR[91,2] = PR[90,2] + -19.259;
   1:L PR[91] R[100]mm/sec CNT100;
   1:  PR[91,1] = PR[90,1] + -73.654;
   1:  PR[91,2] = PR[90,2] + -19.475;
   1:L PR[91] R[100]mm/sec CNT100;
   1:  PR[91,1] = PR[90,1] + -70.925;
   1:  PR[91,2] = PR[90,2] + -19.535;
   1:L PR[91] R[100]mm/sec CNT100;
   1:  PR[91,1] = PR[90,1] + -69.472;
   1:  PR[91,2] = PR[90,2] + -19.588;
   1:L PR[91] R[100]mm/sec CNT100;
   1:  PR[91,1] = PR[90,1] + -67.329;
   1:  PR[91,2] = PR[90,2] + -19.205;
   1:L PR[91] R[100]mm/sec CNT100;
   1:  PR[91,1] = PR[90,1] + -65.328;
   1:  PR[91,2] = PR[90,2] + -18.879;
   1:L PR[91] R[100]mm/sec CNT100;
   1:  PR[91,1] = PR[90,1] + -63.871;
   1:  PR[91,2] = PR[90,2] + -18.299;
   1:L PR[91] R[100]mm/sec CNT100;
   1:  PR[91,1] = PR[90,1] + -61.406;
   1:  PR[91,2] = PR[90,2] + -17.361;
   1:L PR[91] R[100]mm/sec CNT100;
   1:  PR[91,1] = PR[90,1] + -60.629;
   1:  PR[91,2] = PR[90,2] + -16.848;
   1:L PR[91] R[100]mm/sec CNT100;
   1:  PR[91,1] = PR[90,1] + -57.871;
   1:  PR[91,2] = PR[90,2] + -15.084;
   1:L PR[91] R[100]mm/sec CNT100;
   1:  PR[91,1] = PR[90,1] + -55.179;
   1:  PR[91,2] = PR[90,2] + -12.403;
   1:L PR[91] R[100]mm/sec CNT100;
   1:  PR[91,1] = PR[90,1] + -54.850;
   1:  PR[91,2] = PR[90,2] + -12.098;
   1:L PR[91] R[100]mm/sec CNT100;
   1:  PR[91,1] = PR[90,1] + -52.476;
   1:  PR[91,2] = PR[90,2] + -8.631;
   1:L PR[91] R[100]mm/sec CNT100;
   1:  PR[91,1] = PR[90,1] + -50.998;
   1:  PR[91,2] = PR[90,2] + -4.779;
   1:L PR[91] R[100]mm/sec CNT100;
   1:  PR[91,1] = PR[90,1] + -50.624;
   1:  PR[91,2] = PR[90,2] + -1.776;
   1:L PR[91] R[100]mm/sec CNT100TB   .50sec,CALL END_PUD;
   1:  PR[92] = PR[91];
   1:  PR[92,3] = PR[92,3] + 20;
   1:J PR[92] 10% FINE;
   1:  PR[91] = PR[90];
   1:  PR[91,1] = PR[90,1] + 4.469;
   1:  PR[91,2] = PR[90,2] + -0.729;
   1:  PR[91,3] = PR[90,3] + 32.695;
   1:  PR[92] = PR[91];
   1:  PR[92,3] = PR[92,3] + 20;
   1:J PR[92] 10% FINE;
   1:L PR[91] R[100]mm/sec CNT100;
   1:  CALL LASER_DRAHT_START;
   1:  PR[91,1] = PR[90,1] + 5.143;
   1:  PR[91,2] = PR[90,2] + -5.829;
   1:L PR[91] R[100]mm/sec CNT100;
   1:  PR[91,1] = PR[90,1] + 7.118;
   1:  PR[91,2] = PR[90,2] + -10.577;
   1:L PR[91] R[100]mm/sec CNT100;
   1:  PR[91,1] = PR[90,1] + 10.256;
   1:  PR[91,2] = PR[90,2] + -14.648;
   1:L PR[91] R[100]mm/sec CNT100;
   1:  PR[91,1] = PR[90,1] + 14.340;
   1:  PR[91,2] = PR[90,2] + -17.763;
   1:L PR[91] R[100]mm/sec CNT100;
   1:  PR[91,1] = PR[90,1] + 17.726;
   1:  PR[91,2] = PR[90,2] + -19.159;
   1:L PR[91] R[100]mm/sec CNT100;
   1:  PR[91,1] = PR[90,1] + 19.081;
   1:  PR[91,2] = PR[90,2] + -19.714;
   1:L PR[91] R[100]mm/sec CNT100;
   1:  PR[91,1] = PR[90,1] + 24.162;
   1:  PR[91,2] = PR[90,2] + -20.375;
   1:L PR[91] R[100]mm/sec CNT100;
   1:  PR[91,1] = PR[90,1] + 29.234;
   1:  PR[91,2] = PR[90,2] + -19.704;
   1:L PR[91] R[100]mm/sec CNT100;
   1:  PR[91,1] = PR[90,1] + 32.324;
   1:  PR[91,2] = PR[90,2] + -18.438;
   1:L PR[91] R[100]mm/sec CNT100;
   1:  PR[91,1] = PR[90,1] + 33.950;
   1:  PR[91,2] = PR[90,2] + -17.758;
   1:L PR[91] R[100]mm/sec CNT100;
   1:  PR[91,1] = PR[90,1] + 36.544;
   1:  PR[91,2] = PR[90,2] + -15.795;
   1:L PR[91] R[100]mm/sec CNT100;
   1:  PR[91,1] = PR[90,1] + 38.003;
   1:  PR[91,2] = PR[90,2] + -14.670;
   1:L PR[91] R[100]mm/sec CNT100;
   1:  PR[91,1] = PR[90,1] + 39.978;
   1:  PR[91,2] = PR[90,2] + -12.142;
   1:L PR[91] R[100]mm/sec CNT100;
   1:  PR[91,1] = PR[90,1] + 41.183;
   1:  PR[91,2] = PR[90,2] + -10.565;
   1:L PR[91] R[100]mm/sec CNT100;
   1:  PR[91,1] = PR[90,1] + 41.364;
   1:  PR[91,2] = PR[90,2] + -10.235;
   1:L PR[91] R[100]mm/sec CNT100;
   1:  PR[91,1] = PR[90,1] + 42.070;
   1:  PR[91,2] = PR[90,2] + -8.524;
   1:L PR[91] R[100]mm/sec CNT100;
   1:  PR[91,1] = PR[90,1] + 42.766;
   1:  PR[91,2] = PR[90,2] + -6.971;
   1:L PR[91] R[100]mm/sec CNT100;
   1:  PR[91,1] = PR[90,1] + 43.473;
   1:  PR[91,2] = PR[90,2] + -4.203;
   1:L PR[91] R[100]mm/sec CNT100;
   1:  PR[91,1] = PR[90,1] + 43.657;
   1:  PR[91,2] = PR[90,2] + -2.266;
   1:L PR[91] R[100]mm/sec CNT100;
   1:  PR[91,1] = PR[90,1] + 47.140;
   1:  PR[91,2] = PR[90,2] + -2.119;
   1:L PR[91] R[100]mm/sec CNT100;
   1:  PR[91,1] = PR[90,1] + 47.551;
   1:  PR[91,2] = PR[90,2] + -4.387;
   1:L PR[91] R[100]mm/sec CNT100;
   1:  PR[91,1] = PR[90,1] + 47.975;
   1:  PR[91,2] = PR[90,2] + -5.947;
   1:L PR[91] R[100]mm/sec CNT100;
   1:  PR[91,1] = PR[90,1] + 48.962;
   1:  PR[91,2] = PR[90,2] + -7.849;
   1:L PR[91] R[100]mm/sec CNT100;
   1:  PR[91,1] = PR[90,1] + 50.226;
   1:  PR[91,2] = PR[90,2] + -10.536;
   1:L PR[91] R[100]mm/sec CNT100;
   1:  PR[91,1] = PR[90,1] + 50.408;
   1:  PR[91,2] = PR[90,2] + -10.773;
   1:L PR[91] R[100]mm/sec CNT100;
   1:  PR[91,1] = PR[90,1] + 53.451;
   1:  PR[91,2] = PR[90,2] + -14.307;
   1:L PR[91] R[100]mm/sec CNT100;
   1:  PR[91,1] = PR[90,1] + 54.867;
   1:  PR[91,2] = PR[90,2] + -15.442;
   1:L PR[91] R[100]mm/sec CNT100;
   1:  PR[91,1] = PR[90,1] + 57.318;
   1:  PR[91,2] = PR[90,2] + -17.146;
   1:L PR[91] R[100]mm/sec CNT100;
   1:  PR[91,1] = PR[90,1] + 60.422;
   1:  PR[91,2] = PR[90,2] + -18.651;
   1:L PR[91] R[100]mm/sec CNT100;
   1:  PR[91,1] = PR[90,1] + 61.529;
   1:  PR[91,2] = PR[90,2] + -19.083;
   1:L PR[91] R[100]mm/sec CNT100;
   1:  PR[91,1] = PR[90,1] + 65.504;
   1:  PR[91,2] = PR[90,2] + -20.053;
   1:L PR[91] R[100]mm/sec CNT100;
   1:  PR[91,1] = PR[90,1] + 66.069;
   1:  PR[91,2] = PR[90,2] + -20.209;
   1:L PR[91] R[100]mm/sec CNT100;
   1:  PR[91,1] = PR[90,1] + 70.771;
   1:  PR[91,2] = PR[90,2] + -20.477;
   1:L PR[91] R[100]mm/sec CNT100;
   1:  PR[91,1] = PR[90,1] + 71.856;
   1:  PR[91,2] = PR[90,2] + -20.322;
   1:L PR[91] R[100]mm/sec CNT100;
   1:  PR[91,1] = PR[90,1] + 75.350;
   1:  PR[91,2] = PR[90,2] + -19.774;
   1:L PR[91] R[100]mm/sec CNT100;
   1:  PR[91,1] = PR[90,1] + 77.247;
   1:  PR[91,2] = PR[90,2] + -19.075;
   1:L PR[91] R[100]mm/sec CNT100;
   1:  PR[91,1] = PR[90,1] + 79.618;
   1:  PR[91,2] = PR[90,2] + -18.166;
   1:L PR[91] R[100]mm/sec CNT100;
   1:  PR[91,1] = PR[90,1] + 81.915;
   1:  PR[91,2] = PR[90,2] + -16.702;
   1:L PR[91] R[100]mm/sec CNT100;
   1:  PR[91,1] = PR[90,1] + 83.382;
   1:  PR[91,2] = PR[90,2] + -15.743;
   1:L PR[91] R[100]mm/sec CNT100;
   1:  PR[91,1] = PR[90,1] + 86.493;
   1:  PR[91,2] = PR[90,2] + -12.622;
   1:L PR[91] R[100]mm/sec CNT100;
   1:  PR[91,1] = PR[90,1] + 88.806;
   1:  PR[91,2] = PR[90,2] + -8.967;
   1:L PR[91] R[100]mm/sec CNT100;
   1:  PR[91,1] = PR[90,1] + 90.231;
   1:  PR[91,2] = PR[90,2] + -4.940;
   1:L PR[91] R[100]mm/sec CNT100;
   1:  PR[91,1] = PR[90,1] + 90.718;
   1:  PR[91,2] = PR[90,2] + -0.729;
   1:L PR[91] R[100]mm/sec CNT100;
   1:  PR[91,1] = PR[90,1] + 90.231;
   1:  PR[91,2] = PR[90,2] + 3.481;
   1:L PR[91] R[100]mm/sec CNT100;
   1:  PR[91,1] = PR[90,1] + 88.806;
   1:  PR[91,2] = PR[90,2] + 7.508;
   1:L PR[91] R[100]mm/sec CNT100;
   1:  PR[91,1] = PR[90,1] + 86.495;
   1:  PR[91,2] = PR[90,2] + 11.160;
   1:L PR[91] R[100]mm/sec CNT100;
   1:  PR[91,1] = PR[90,1] + 84.284;
   1:  PR[91,2] = PR[90,2] + 13.362;
   1:L PR[91] R[100]mm/sec CNT100;
   1:  PR[91,1] = PR[90,1] + 83.384;
   1:  PR[91,2] = PR[90,2] + 14.279;
   1:L PR[91] R[100]mm/sec CNT100;
   1:  PR[91,1] = PR[90,1] + 81.098;
   1:  PR[91,2] = PR[90,2] + 15.732;
   1:L PR[91] R[100]mm/sec CNT100;
   1:  PR[91,1] = PR[90,1] + 79.618;
   1:  PR[91,2] = PR[90,2] + 16.704;
   1:L PR[91] R[100]mm/sec CNT100;
   1:  PR[91,1] = PR[90,1] + 77.562;
   1:  PR[91,2] = PR[90,2] + 17.457;
   1:L PR[91] R[100]mm/sec CNT100;
   1:  PR[91,1] = PR[90,1] + 75.350;
   1:  PR[91,2] = PR[90,2] + 18.312;
   1:L PR[91] R[100]mm/sec CNT100;
   1:  PR[91,1] = PR[90,1] + 73.814;
   1:  PR[91,2] = PR[90,2] + 18.527;
   1:L PR[91] R[100]mm/sec CNT100;
   1:  PR[91,1] = PR[90,1] + 70.770;
   1:  PR[91,2] = PR[90,2] + 19.014;
   1:L PR[91] R[100]mm/sec CNT100;
   1:  PR[91,1] = PR[90,1] + 69.982;
   1:  PR[91,2] = PR[90,2] + 18.956;
   1:L PR[91] R[100]mm/sec CNT100;
   1:  PR[91,1] = PR[90,1] + 66.065;
   1:  PR[91,2] = PR[90,2] + 18.749;
   1:L PR[91] R[100]mm/sec CNT100;
   1:  PR[91,1] = PR[90,1] + 65.504;
   1:  PR[91,2] = PR[90,2] + 18.594;
   1:L PR[91] R[100]mm/sec CNT100;
   1:  PR[91,1] = PR[90,1] + 61.529;
   1:  PR[91,2] = PR[90,2] + 17.625;
   1:L PR[91] R[100]mm/sec CNT100;
   1:  PR[91,1] = PR[90,1] + 60.422;
   1:  PR[91,2] = PR[90,2] + 17.192;
   1:L PR[91] R[100]mm/sec CNT100;
   1:  PR[91,1] = PR[90,1] + 57.318;
   1:  PR[91,2] = PR[90,2] + 15.687;
   1:L PR[91] R[100]mm/sec CNT100;
   1:  PR[91,1] = PR[90,1] + 54.868;
   1:  PR[91,2] = PR[90,2] + 13.984;
   1:L PR[91] R[100]mm/sec CNT100;
   1:  PR[91,1] = PR[90,1] + 53.452;
   1:  PR[91,2] = PR[90,2] + 12.849;
   1:L PR[91] R[100]mm/sec CNT100;
   1:  PR[91,1] = PR[90,1] + 50.409;
   1:  PR[91,2] = PR[90,2] + 9.316;
   1:L PR[91] R[100]mm/sec CNT100;
   1:  PR[91,1] = PR[90,1] + 50.226;
   1:  PR[91,2] = PR[90,2] + 9.078;
   1:L PR[91] R[100]mm/sec CNT100;
   1:  PR[91,1] = PR[90,1] + 48.961;
   1:  PR[91,2] = PR[90,2] + 6.389;
   1:L PR[91] R[100]mm/sec CNT100;
   1:  PR[91,1] = PR[90,1] + 47.985;
   1:  PR[91,2] = PR[90,2] + 4.511;
   1:L PR[91] R[100]mm/sec CNT100;
   1:  PR[91,1] = PR[90,1] + 47.482;
   1:  PR[91,2] = PR[90,2] + 2.646;
   1:L PR[91] R[100]mm/sec CNT100;
   1:  PR[91,1] = PR[90,1] + 47.137;
   1:  PR[91,2] = PR[90,2] + 0.760;
   1:L PR[91] R[100]mm/sec CNT100;
   1:  PR[91,1] = PR[90,1] + 43.653;
   1:  PR[91,2] = PR[90,2] + 0.914;
   1:L PR[91] R[100]mm/sec CNT100;
   1:  PR[91,1] = PR[90,1] + 43.495;
   1:  PR[91,2] = PR[90,2] + 2.623;
   1:L PR[91] R[100]mm/sec CNT100;
   1:  PR[91,1] = PR[90,1] + 42.693;
   1:  PR[91,2] = PR[90,2] + 5.724;
   1:L PR[91] R[100]mm/sec CNT100;
   1:  PR[91,1] = PR[90,1] + 42.326;
   1:  PR[91,2] = PR[90,2] + 6.613;
   1:L PR[91] R[100]mm/sec CNT100;
   1:  PR[91,1] = PR[90,1] + 41.404;
   1:  PR[91,2] = PR[90,2] + 8.700;
   1:L PR[91] R[100]mm/sec CNT100;
   1:  PR[91,1] = PR[90,1] + 41.184;
   1:  PR[91,2] = PR[90,2] + 9.104;
   1:L PR[91] R[100]mm/sec CNT100;
   1:  PR[91,1] = PR[90,1] + 39.948;
   1:  PR[91,2] = PR[90,2] + 10.732;
   1:L PR[91] R[100]mm/sec CNT100;
   1:  PR[91,1] = PR[90,1] + 37.982;
   1:  PR[91,2] = PR[90,2] + 13.232;
   1:L PR[91] R[100]mm/sec CNT100;
   1:  PR[91,1] = PR[90,1] + 36.524;
   1:  PR[91,2] = PR[90,2] + 14.357;
   1:L PR[91] R[100]mm/sec CNT100;
   1:  PR[91,1] = PR[90,1] + 33.926;
   1:  PR[91,2] = PR[90,2] + 16.313;
   1:L PR[91] R[100]mm/sec CNT100;
   1:  PR[91,1] = PR[90,1] + 32.300;
   1:  PR[91,2] = PR[90,2] + 16.993;
   1:L PR[91] R[100]mm/sec CNT100;
   1:  PR[91,1] = PR[90,1] + 29.208;
   1:  PR[91,2] = PR[90,2] + 18.253;
   1:L PR[91] R[100]mm/sec CNT100;
   1:  PR[91,1] = PR[90,1] + 27.552;
   1:  PR[91,2] = PR[90,2] + 18.478;
   1:L PR[91] R[100]mm/sec CNT100;
   1:  PR[91,1] = PR[90,1] + 24.143;
   1:  PR[91,2] = PR[90,2] + 18.917;
   1:L PR[91] R[100]mm/sec CNT100;
   1:  PR[91,1] = PR[90,1] + 19.065;
   1:  PR[91,2] = PR[90,2] + 18.251;
   1:L PR[91] R[100]mm/sec CNT100;
   1:  PR[91,1] = PR[90,1] + 14.324;
   1:  PR[91,2] = PR[90,2] + 16.295;
   1:L PR[91] R[100]mm/sec CNT100;
   1:  PR[91,1] = PR[90,1] + 13.237;
   1:  PR[91,2] = PR[90,2] + 15.467;
   1:L PR[91] R[100]mm/sec CNT100;
   1:  PR[91,1] = PR[90,1] + 10.248;
   1:  PR[91,2] = PR[90,2] + 13.181;
   1:L PR[91] R[100]mm/sec CNT100;
   1:  PR[91,1] = PR[90,1] + 7.114;
   1:  PR[91,2] = PR[90,2] + 9.111;
   1:L PR[91] R[100]mm/sec CNT100;
   1:  PR[91,1] = PR[90,1] + 5.142;
   1:  PR[91,2] = PR[90,2] + 4.367;
   1:L PR[91] R[100]mm/sec CNT100;
   1:  PR[91,1] = PR[90,1] + 4.469;
   1:  PR[91,2] = PR[90,2] + -0.729;
   1:L PR[91] R[100]mm/sec CNT100TB   .50sec,CALL END_PUD;
   1:  PR[92] = PR[91];
   1:  PR[92,3] = PR[92,3] + 20;
   1:J PR[92] 10% FINE;
   1:  PR[91,1] = PR[90,1] + -41.681;
   1:  PR[91,2] = PR[90,2] + -0.717;
   1:  PR[92] = PR[91];
   1:  PR[92,3] = PR[92,3] + 20;
   1:J PR[92] 10% FINE;
   1:L PR[91] R[100]mm/sec CNT100;
   1:  CALL LASER_DRAHT_START;
   1:  PR[91,1] = PR[90,1] + -41.546;
   1:  PR[91,2] = PR[90,2] + -1.807;
   1:L PR[91] R[100]mm/sec CNT100;
   1:  PR[91,1] = PR[90,1] + -41.199;
   1:  PR[91,2] = PR[90,2] + -4.905;
   1:L PR[91] R[100]mm/sec CNT100;
   1:  PR[91,1] = PR[90,1] + -39.815;
   1:  PR[91,2] = PR[90,2] + -8.880;
   1:L PR[91] R[100]mm/sec CNT100;
   1:  PR[91,1] = PR[90,1] + -37.577;
   1:  PR[91,2] = PR[90,2] + -12.464;
   1:L PR[91] R[100]mm/sec CNT100;
   1:  PR[91,1] = PR[90,1] + -34.591;
   1:  PR[91,2] = PR[90,2] + -15.481;
   1:L PR[91] R[100]mm/sec CNT100;
   1:  PR[91,1] = PR[90,1] + -30.997;
   1:  PR[91,2] = PR[90,2] + -17.783;
   1:L PR[91] R[100]mm/sec CNT100;
   1:  PR[91,1] = PR[90,1] + -26.963;
   1:  PR[91,2] = PR[90,2] + -19.248;
   1:L PR[91] R[100]mm/sec CNT100;
   1:  PR[91,1] = PR[90,1] + -22.671;
   1:  PR[91,2] = PR[90,2] + -19.803;
   1:L PR[91] R[100]mm/sec CNT100;
   1:  PR[91,1] = PR[90,1] + -18.279;
   1:  PR[91,2] = PR[90,2] + -19.439;
   1:L PR[91] R[100]mm/sec CNT100;
   1:  PR[91,1] = PR[90,1] + -18.066;
   1:  PR[91,2] = PR[90,2] + -19.387;
   1:L PR[91] R[100]mm/sec CNT100;
   1:  PR[91,1] = PR[90,1] + -14.122;
   1:  PR[91,2] = PR[90,2] + -18.164;
   1:L PR[91] R[100]mm/sec CNT100;
   1:  PR[91,1] = PR[90,1] + -13.522;
   1:  PR[91,2] = PR[90,2] + -17.867;
   1:L PR[91] R[100]mm/sec CNT100;
   1:  PR[91,1] = PR[90,1] + -10.339;
   1:  PR[91,2] = PR[90,2] + -16.033;
   1:L PR[91] R[100]mm/sec CNT100;
   1:  PR[91,1] = PR[90,1] + -9.487;
   1:  PR[91,2] = PR[90,2] + -15.341;
   1:L PR[91] R[100]mm/sec CNT100;
   1:  PR[91,1] = PR[90,1] + -7.115;
   1:  PR[91,2] = PR[90,2] + -13.139;
   1:L PR[91] R[100]mm/sec CNT100;
   1:  PR[91,1] = PR[90,1] + -6.219;
   1:  PR[91,2] = PR[90,2] + -11.981;
   1:L PR[91] R[100]mm/sec CNT100;
   1:  PR[91,1] = PR[90,1] + -4.619;
   1:  PR[91,2] = PR[90,2] + -9.603;
   1:L PR[91] R[100]mm/sec CNT100;
   1:  PR[91,1] = PR[90,1] + -3.902;
   1:  PR[91,2] = PR[90,2] + -8.021;
   1:L PR[91] R[100]mm/sec CNT100;
   1:  PR[91,1] = PR[90,1] + -2.996;
   1:  PR[91,2] = PR[90,2] + -5.591;
   1:L PR[91] R[100]mm/sec CNT100;
   1:  PR[91,1] = PR[90,1] + -2.643;
   1:  PR[91,2] = PR[90,2] + -3.715;
   1:L PR[91] R[100]mm/sec CNT100;
   1:  PR[91,1] = PR[90,1] + -2.344;
   1:  PR[91,2] = PR[90,2] + -1.237;
   1:L PR[91] R[100]mm/sec CNT100;
   1:  PR[91,1] = PR[90,1] + -2.332;
   1:  PR[91,2] = PR[90,2] + -0.821;
   1:L PR[91] R[100]mm/sec CNT100;
   1:  PR[91,1] = PR[90,1] + -2.639;
   1:  PR[91,2] = PR[90,2] + 1.729;
   1:L PR[91] R[100]mm/sec CNT100;
   1:  PR[91,1] = PR[90,1] + -2.659;
   1:  PR[91,2] = PR[90,2] + 2.337;
   1:L PR[91] R[100]mm/sec CNT100;
   1:  PR[91,1] = PR[90,1] + -2.994;
   1:  PR[91,2] = PR[90,2] + 4.125;
   1:L PR[91] R[100]mm/sec CNT100;
   1:  PR[91,1] = PR[90,1] + -3.900;
   1:  PR[91,2] = PR[90,2] + 6.556;
   1:L PR[91] R[100]mm/sec CNT100;
   1:  PR[91,1] = PR[90,1] + -4.616;
   1:  PR[91,2] = PR[90,2] + 8.139;
   1:L PR[91] R[100]mm/sec CNT100;
   1:  PR[91,1] = PR[90,1] + -6.216;
   1:  PR[91,2] = PR[90,2] + 10.518;
   1:L PR[91] R[100]mm/sec CNT100;
   1:  PR[91,1] = PR[90,1] + -7.112;
   1:  PR[91,2] = PR[90,2] + 11.677;
   1:L PR[91] R[100]mm/sec CNT100;
   1:  PR[91,1] = PR[90,1] + -9.484;
   1:  PR[91,2] = PR[90,2] + 13.879;
   1:L PR[91] R[100]mm/sec CNT100;
   1:  PR[91,1] = PR[90,1] + -10.336;
   1:  PR[91,2] = PR[90,2] + 14.573;
   1:L PR[91] R[100]mm/sec CNT100;
   1:  PR[91,1] = PR[90,1] + -13.520;
   1:  PR[91,2] = PR[90,2] + 16.407;
   1:L PR[91] R[100]mm/sec CNT100;
   1:  PR[91,1] = PR[90,1] + -14.120;
   1:  PR[91,2] = PR[90,2] + 16.705;
   1:L PR[91] R[100]mm/sec CNT100;
   1:  PR[91,1] = PR[90,1] + -18.065;
   1:  PR[91,2] = PR[90,2] + 17.927;
   1:L PR[91] R[100]mm/sec CNT100;
   1:  PR[91,1] = PR[90,1] + -18.278;
   1:  PR[91,2] = PR[90,2] + 17.980;
   1:L PR[91] R[100]mm/sec CNT100;
   1:  PR[91,1] = PR[90,1] + -22.679;
   1:  PR[91,2] = PR[90,2] + 18.344;
   1:L PR[91] R[100]mm/sec CNT100;
   1:  PR[91,1] = PR[90,1] + -26.963;
   1:  PR[91,2] = PR[90,2] + 17.790;
   1:L PR[91] R[100]mm/sec CNT100;
   1:  PR[91,1] = PR[90,1] + -30.997;
   1:  PR[91,2] = PR[90,2] + 16.324;
   1:L PR[91] R[100]mm/sec CNT100;
   1:  PR[91,1] = PR[90,1] + -34.591;
   1:  PR[91,2] = PR[90,2] + 14.022;
   1:L PR[91] R[100]mm/sec CNT100;
   1:  PR[91,1] = PR[90,1] + -37.577;
   1:  PR[91,2] = PR[90,2] + 11.005;
   1:L PR[91] R[100]mm/sec CNT100;
   1:  PR[91,1] = PR[90,1] + -39.815;
   1:  PR[91,2] = PR[90,2] + 7.422;
   1:L PR[91] R[100]mm/sec CNT100;
   1:  PR[91,1] = PR[90,1] + -41.199;
   1:  PR[91,2] = PR[90,2] + 3.445;
   1:L PR[91] R[100]mm/sec CNT100;
   1:  PR[91,1] = PR[90,1] + -41.330;
   1:  PR[91,2] = PR[90,2] + 2.291;
   1:L PR[91] R[100]mm/sec CNT100;
   1:  PR[91,1] = PR[90,1] + -41.361;
   1:  PR[91,2] = PR[90,2] + 2.140;
   1:L PR[91] R[100]mm/sec CNT100;
   1:  PR[91,1] = PR[90,1] + -41.681;
   1:  PR[91,2] = PR[90,2] + -0.717;
   1:L PR[91] R[100]mm/sec CNT100TB   .50sec,CALL END_PUD;
   1:  PR[92] = PR[91];
   1:  PR[92,3] = PR[92,3] + 20;
   1:J PR[92] 10% FINE;
   1:  PR[91,1] = PR[90,1] + -77.314;
   1:  PR[91,2] = PR[90,2] + -18.642;
   1:  PR[92] = PR[91];
   1:  PR[92,3] = PR[92,3] + 20;
   1:J PR[92] 10% FINE;
   1:L PR[91] R[100]mm/sec CNT100;
   1:  CALL LASER_DRAHT_START;
   1:  PR[91,1] = PR[90,1] + -74.683;
   1:  PR[91,2] = PR[90,2] + -19.231;
   1:L PR[91] R[100]mm/sec CNT100;
   1:  PR[91,1] = PR[90,1] + -73.251;
   1:  PR[91,2] = PR[90,2] + -19.573;
   1:L PR[91] R[100]mm/sec CNT100;
   1:  PR[91,1] = PR[90,1] + -71.069;
   1:  PR[91,2] = PR[90,2] + -19.621;
   1:L PR[91] R[100]mm/sec CNT100;
   1:  PR[91,1] = PR[90,1] + -69.047;
   1:  PR[91,2] = PR[90,2] + -19.694;
   1:L PR[91] R[100]mm/sec CNT100;
   1:  PR[91,1] = PR[90,1] + -67.474;
   1:  PR[91,2] = PR[90,2] + -19.413;
   1:L PR[91] R[100]mm/sec CNT100;
   1:  PR[91,1] = PR[90,1] + -64.878;
   1:  PR[91,2] = PR[90,2] + -18.989;
   1:L PR[91] R[100]mm/sec CNT100;
   1:  PR[91,1] = PR[90,1] + -63.990;
   1:  PR[91,2] = PR[90,2] + -18.636;
   1:L PR[91] R[100]mm/sec CNT100;
   1:  PR[91,1] = PR[90,1] + -60.914;
   1:  PR[91,2] = PR[90,2] + -17.467;
   1:L PR[91] R[100]mm/sec CNT100;
   1:  PR[91,1] = PR[90,1] + -58.205;
   1:  PR[91,2] = PR[90,2] + -15.726;
   1:L PR[91] R[100]mm/sec CNT100;
   1:  PR[91,1] = PR[90,1] + -57.250;
   1:  PR[91,2] = PR[90,2] + -15.156;
   1:L PR[91] R[100]mm/sec CNT100;
   1:  PR[91,1] = PR[90,1] + -54.565;
   1:  PR[91,2] = PR[90,2] + -12.649;
   1:L PR[91] R[100]mm/sec CNT100;
   1:  PR[91,1] = PR[90,1] + -54.071;
   1:  PR[91,2] = PR[90,2] + -12.203;
   1:L PR[91] R[100]mm/sec CNT100;
   1:  PR[91,1] = PR[90,1] + -52.386;
   1:  PR[91,2] = PR[90,2] + -9.733;
   1:L PR[91] R[100]mm/sec CNT100;
   1:  PR[91,1] = PR[90,1] + -51.665;
   1:  PR[91,2] = PR[90,2] + -8.704;
   1:L PR[91] R[100]mm/sec CNT100;
   1:  PR[91,1] = PR[90,1] + -50.168;
   1:  PR[91,2] = PR[90,2] + -4.823;
   1:L PR[91] R[100]mm/sec CNT100;
   1:  PR[91,1] = PR[90,1] + -49.910;
   1:  PR[91,2] = PR[90,2] + -2.744;
   1:L PR[91] R[100]mm/sec CNT100;
   1:  PR[91,1] = PR[90,1] + -49.770;
   1:  PR[91,2] = PR[90,2] + -0.743;
   1:L PR[91] R[100]mm/sec CNT100;
   1:  PR[91,1] = PR[90,1] + -49.798;
   1:  PR[91,2] = PR[90,2] + -0.406;
   1:L PR[91] R[100]mm/sec CNT100;
   1:  PR[91,1] = PR[90,1] + -50.252;
   1:  PR[91,2] = PR[90,2] + 3.373;
   1:L PR[91] R[100]mm/sec CNT100;
   1:  PR[91,1] = PR[90,1] + -51.720;
   1:  PR[91,2] = PR[90,2] + 7.273;
   1:L PR[91] R[100]mm/sec CNT100;
   1:  PR[91,1] = PR[90,1] + -52.373;
   1:  PR[91,2] = PR[90,2] + 8.257;
   1:L PR[91] R[100]mm/sec CNT100;
   1:  PR[91,1] = PR[90,1] + -54.073;
   1:  PR[91,2] = PR[90,2] + 10.775;
   1:L PR[91] R[100]mm/sec CNT100;
   1:  PR[91,1] = PR[90,1] + -55.593;
   1:  PR[91,2] = PR[90,2] + 12.234;
   1:L PR[91] R[100]mm/sec CNT100;
   1:  PR[91,1] = PR[90,1] + -57.173;
   1:  PR[91,2] = PR[90,2] + 13.722;
   1:L PR[91] R[100]mm/sec CNT100;
   1:  PR[91,1] = PR[90,1] + -60.872;
   1:  PR[91,2] = PR[90,2] + 15.996;
   1:L PR[91] R[100]mm/sec CNT100;
   1:  PR[91,1] = PR[90,1] + -64.984;
   1:  PR[91,2] = PR[90,2] + 17.505;
   1:L PR[91] R[100]mm/sec CNT100;
   1:  PR[91,1] = PR[90,1] + -69.137;
   1:  PR[91,2] = PR[90,2] + 18.221;
   1:L PR[91] R[100]mm/sec CNT100;
   1:  PR[91,1] = PR[90,1] + -73.297;
   1:  PR[91,2] = PR[90,2] + 18.107;
   1:L PR[91] R[100]mm/sec CNT100;
   1:  PR[91,1] = PR[90,1] + -77.320;
   1:  PR[91,2] = PR[90,2] + 17.184;
   1:L PR[91] R[100]mm/sec CNT100;
   1:  PR[91,1] = PR[90,1] + -81.037;
   1:  PR[91,2] = PR[90,2] + 15.500;
   1:L PR[91] R[100]mm/sec CNT100;
   1:  PR[91,1] = PR[90,1] + -84.300;
   1:  PR[91,2] = PR[90,2] + 13.138;
   1:L PR[91] R[100]mm/sec CNT100;
   1:  PR[91,1] = PR[90,1] + -86.977;
   1:  PR[91,2] = PR[90,2] + 10.199;
   1:L PR[91] R[100]mm/sec CNT100;
   1:  PR[91,1] = PR[90,1] + -88.967;
   1:  PR[91,2] = PR[90,2] + 6.813;
   1:L PR[91] R[100]mm/sec CNT100;
   1:  PR[91,1] = PR[90,1] + -90.190;
   1:  PR[91,2] = PR[90,2] + 3.119;
   1:L PR[91] R[100]mm/sec CNT100;
   1:  PR[91,1] = PR[90,1] + -90.556;
   1:  PR[91,2] = PR[90,2] + -0.259;
   1:L PR[91] R[100]mm/sec CNT100;
   1:  PR[91,1] = PR[90,1] + -90.654;
   1:  PR[91,2] = PR[90,2] + -0.746;
   1:L PR[91] R[100]mm/sec CNT100;
   1:  PR[91,1] = PR[90,1] + -90.252;
   1:  PR[91,2] = PR[90,2] + -4.584;
   1:L PR[91] R[100]mm/sec CNT100;
   1:  PR[91,1] = PR[90,1] + -89.055;
   1:  PR[91,2] = PR[90,2] + -8.268;
   1:L PR[91] R[100]mm/sec CNT100;
   1:  PR[91,1] = PR[90,1] + -87.060;
   1:  PR[91,2] = PR[90,2] + -11.645;
   1:L PR[91] R[100]mm/sec CNT100;
   1:  PR[91,1] = PR[90,1] + -84.363;
   1:  PR[91,2] = PR[90,2] + -14.584;
   1:L PR[91] R[100]mm/sec CNT100;
   1:  PR[91,1] = PR[90,1] + -81.074;
   1:  PR[91,2] = PR[90,2] + -16.950;
   1:L PR[91] R[100]mm/sec CNT100;
   1:  PR[91,1] = PR[90,1] + -78.209;
   1:  PR[91,2] = PR[90,2] + -18.229;
   1:L PR[91] R[100]mm/sec CNT100;
   1:  PR[91,1] = PR[90,1] + -77.314;
   1:  PR[91,2] = PR[90,2] + -18.642;
   1:L PR[91] R[100]mm/sec CNT100TB   .50sec,CALL END_PUD;
   1:  PR[92] = PR[91];
   1:  PR[92,3] = PR[92,3] + 20;
   1:J PR[92] 10% FINE;
   1:  PR[91] = PR[90];
   1:  PR[91,1] = PR[90,1] + 4.937;
   1:  PR[91,2] = PR[90,2] + -5.866;
   1:  PR[91,3] = PR[90,3] + 33.995;
   1:  PR[92] = PR[91];
   1:  PR[92,3] = PR[92,3] + 20;
   1:J PR[92] 10% FINE;
   1:L PR[91] R[100]mm/sec CNT100;
   1:  CALL LASER_DRAHT_START;
   1:  PR[91,1] = PR[90,1] + 6.927;
   1:  PR[91,2] = PR[90,2] + -10.647;
   1:L PR[91] R[100]mm/sec CNT100;
   1:  PR[91,1] = PR[90,1] + 10.086;
   1:  PR[91,2] = PR[90,2] + -14.747;
   1:L PR[91] R[100]mm/sec CNT100;
   1:  PR[91,1] = PR[90,1] + 14.198;
   1:  PR[91,2] = PR[90,2] + -17.884;
   1:L PR[91] R[100]mm/sec CNT100;
   1:  PR[91,1] = PR[90,1] + 18.974;
   1:  PR[91,2] = PR[90,2] + -19.851;
   1:L PR[91] R[100]mm/sec CNT100;
   1:  PR[91,1] = PR[90,1] + 24.089;
   1:  PR[91,2] = PR[90,2] + -20.518;
   1:L PR[91] R[100]mm/sec CNT100;
   1:  PR[91,1] = PR[90,1] + 28.004;
   1:  PR[91,2] = PR[90,2] + -20.007;
   1:L PR[91] R[100]mm/sec CNT100;
   1:  PR[91,1] = PR[90,1] + 29.188;
   1:  PR[91,2] = PR[90,2] + -19.846;
   1:L PR[91] R[100]mm/sec CNT100;
   1:  PR[91,1] = PR[90,1] + 33.946;
   1:  PR[91,2] = PR[90,2] + -17.886;
   1:L PR[91] R[100]mm/sec CNT100;
   1:  PR[91,1] = PR[90,1] + 36.932;
   1:  PR[91,2] = PR[90,2] + -15.626;
   1:L PR[91] R[100]mm/sec CNT100;
   1:  PR[91,1] = PR[90,1] + 38.023;
   1:  PR[91,2] = PR[90,2] + -14.784;
   1:L PR[91] R[100]mm/sec CNT100;
   1:  PR[91,1] = PR[90,1] + 40.305;
   1:  PR[91,2] = PR[90,2] + -11.865;
   1:L PR[91] R[100]mm/sec CNT100;
   1:  PR[91,1] = PR[90,1] + 41.228;
   1:  PR[91,2] = PR[90,2] + -10.656;
   1:L PR[91] R[100]mm/sec CNT100;
   1:  PR[91,1] = PR[90,1] + 41.454;
   1:  PR[91,2] = PR[90,2] + -10.245;
   1:L PR[91] R[100]mm/sec CNT100;
   1:  PR[91,1] = PR[90,1] + 41.969;
   1:  PR[91,2] = PR[90,2] + -8.998;
   1:L PR[91] R[100]mm/sec CNT100;
   1:  PR[91,1] = PR[90,1] + 42.774;
   1:  PR[91,2] = PR[90,2] + -7.199;
   1:L PR[91] R[100]mm/sec CNT100;
   1:  PR[91,1] = PR[90,1] + 44.425;
   1:  PR[91,2] = PR[90,2] + -0.731;
   1:L PR[91] R[100]mm/sec CNT100;
   1:  PR[91,1] = PR[90,1] + 42.691;
   1:  PR[91,2] = PR[90,2] + 5.979;
   1:L PR[91] R[100]mm/sec CNT100;
   1:  PR[91,1] = PR[90,1] + 42.559;
   1:  PR[91,2] = PR[90,2] + 6.299;
   1:L PR[91] R[100]mm/sec CNT100;
   1:  PR[91,1] = PR[90,1] + 41.498;
   1:  PR[91,2] = PR[90,2] + 8.701;
   1:L PR[91] R[100]mm/sec CNT100;
   1:  PR[91,1] = PR[90,1] + 41.229;
   1:  PR[91,2] = PR[90,2] + 9.195;
   1:L PR[91] R[100]mm/sec CNT100;
   1:  PR[91,1] = PR[90,1] + 40.269;
   1:  PR[91,2] = PR[90,2] + 10.462;
   1:L PR[91] R[100]mm/sec CNT100;
   1:  PR[91,1] = PR[90,1] + 37.999;
   1:  PR[91,2] = PR[90,2] + 13.349;
   1:L PR[91] R[100]mm/sec CNT100;
   1:  PR[91,1] = PR[90,1] + 36.907;
   1:  PR[91,2] = PR[90,2] + 14.192;
   1:L PR[91] R[100]mm/sec CNT100;
   1:  PR[91,1] = PR[90,1] + 33.914;
   1:  PR[91,2] = PR[90,2] + 16.446;
   1:L PR[91] R[100]mm/sec CNT100;
   1:  PR[91,1] = PR[90,1] + 32.719;
   1:  PR[91,2] = PR[90,2] + 16.946;
   1:L PR[91] R[100]mm/sec CNT100;
   1:  PR[91,1] = PR[90,1] + 29.163;
   1:  PR[91,2] = PR[90,2] + 18.395;
   1:L PR[91] R[100]mm/sec CNT100;
   1:  PR[91,1] = PR[90,1] + 27.976;
   1:  PR[91,2] = PR[90,2] + 18.556;
   1:L PR[91] R[100]mm/sec CNT100;
   1:  PR[91,1] = PR[90,1] + 24.065;
   1:  PR[91,2] = PR[90,2] + 19.059;
   1:L PR[91] R[100]mm/sec CNT100;
   1:  PR[91,1] = PR[90,1] + 18.954;
   1:  PR[91,2] = PR[90,2] + 18.386;
   1:L PR[91] R[100]mm/sec CNT100;
   1:  PR[91,1] = PR[90,1] + 14.183;
   1:  PR[91,2] = PR[90,2] + 16.417;
   1:L PR[91] R[100]mm/sec CNT100;
   1:  PR[91,1] = PR[90,1] + 10.077;
   1:  PR[91,2] = PR[90,2] + 13.279;
   1:L PR[91] R[100]mm/sec CNT100;
   1:  PR[91,1] = PR[90,1] + 6.922;
   1:  PR[91,2] = PR[90,2] + 9.181;
   1:L PR[91] R[100]mm/sec CNT100;
   1:  PR[91,1] = PR[90,1] + 4.936;
   1:  PR[91,2] = PR[90,2] + 4.403;
   1:L PR[91] R[100]mm/sec CNT100;
   1:  PR[91,1] = PR[90,1] + 4.259;
   1:  PR[91,2] = PR[90,2] + -0.729;
   1:L PR[91] R[100]mm/sec CNT100;
   1:  PR[91,1] = PR[90,1] + 4.937;
   1:  PR[91,2] = PR[90,2] + -5.866;
   1:L PR[91] R[100]mm/sec CNT100TB   .50sec,CALL END_PUD;
   1:  PR[92] = PR[91];
   1:  PR[92,3] = PR[92,3] + 20;
   1:J PR[92] 10% FINE;
   1:  PR[91,1] = PR[90,1] + 45.494;
   1:  PR[91,2] = PR[90,2] + -0.780;
   1:  PR[92] = PR[91];
   1:  PR[92,3] = PR[92,3] + 20;
   1:J PR[92] 10% FINE;
   1:L PR[91] R[100]mm/sec CNT100;
   1:  CALL LASER_DRAHT_START;
   1:  PR[91,1] = PR[90,1] + 47.117;
   1:  PR[91,2] = PR[90,2] + -6.749;
   1:L PR[91] R[100]mm/sec CNT100;
   1:  PR[91,1] = PR[90,1] + 49.050;
   1:  PR[91,2] = PR[90,2] + -10.476;
   1:L PR[91] R[100]mm/sec CNT100;
   1:  PR[91,1] = PR[90,1] + 49.408;
   1:  PR[91,2] = PR[90,2] + -10.911;
   1:L PR[91] R[100]mm/sec CNT100;
   1:  PR[91,1] = PR[90,1] + 51.186;
   1:  PR[91,2] = PR[90,2] + -12.768;
   1:L PR[91] R[100]mm/sec CNT100;
   1:  PR[91,1] = PR[90,1] + 52.835;
   1:  PR[91,2] = PR[90,2] + -14.684;
   1:L PR[91] R[100]mm/sec CNT100;
   1:  PR[91,1] = PR[90,1] + 53.211;
   1:  PR[91,2] = PR[90,2] + -14.985;
   1:L PR[91] R[100]mm/sec CNT100;
   1:  PR[91,1] = PR[90,1] + 56.860;
   1:  PR[91,2] = PR[90,2] + -17.522;
   1:L PR[91] R[100]mm/sec CNT100;
   1:  PR[91,1] = PR[90,1] + 58.877;
   1:  PR[91,2] = PR[90,2] + -18.500;
   1:L PR[91] R[100]mm/sec CNT100;
   1:  PR[91,1] = PR[90,1] + 61.208;
   1:  PR[91,2] = PR[90,2] + -19.410;
   1:L PR[91] R[100]mm/sec CNT100;
   1:  PR[91,1] = PR[90,1] + 64.943;
   1:  PR[91,2] = PR[90,2] + -20.322;
   1:L PR[91] R[100]mm/sec CNT100;
   1:  PR[91,1] = PR[90,1] + 65.668;
   1:  PR[91,2] = PR[90,2] + -20.430;
   1:L PR[91] R[100]mm/sec CNT100;
   1:  PR[91,1] = PR[90,1] + 68.583;
   1:  PR[91,2] = PR[90,2] + -20.534;
   1:L PR[91] R[100]mm/sec CNT100;
   1:  PR[91,1] = PR[90,1] + 70.360;
   1:  PR[91,2] = PR[90,2] + -20.634;
   1:L PR[91] R[100]mm/sec CNT100;
   1:  PR[91,1] = PR[90,1] + 74.988;
   1:  PR[91,2] = PR[90,2] + -19.914;
   1:L PR[91] R[100]mm/sec CNT100;
   1:  PR[91,1] = PR[90,1] + 76.141;
   1:  PR[91,2] = PR[90,2] + -19.489;
   1:L PR[91] R[100]mm/sec CNT100;
   1:  PR[91,1] = PR[90,1] + 79.280;
   1:  PR[91,2] = PR[90,2] + -18.285;
   1:L PR[91] R[100]mm/sec CNT100;
   1:  PR[91,1] = PR[90,1] + 80.968;
   1:  PR[91,2] = PR[90,2] + -17.210;
   1:L PR[91] R[100]mm/sec CNT100;
   1:  PR[91,1] = PR[90,1] + 83.067;
   1:  PR[91,2] = PR[90,2] + -15.837;
   1:L PR[91] R[100]mm/sec CNT100;
   1:  PR[91,1] = PR[90,1] + 84.877;
   1:  PR[91,2] = PR[90,2] + -14.031;
   1:L PR[91] R[100]mm/sec CNT100;
   1:  PR[91,1] = PR[90,1] + 86.185;
   1:  PR[91,2] = PR[90,2] + -12.701;
   1:L PR[91] R[100]mm/sec CNT100;
   1:  PR[91,1] = PR[90,1] + 88.511;
   1:  PR[91,2] = PR[90,2] + -9.016;
   1:L PR[91] R[100]mm/sec CNT100;
   1:  PR[91,1] = PR[90,1] + 89.942;
   1:  PR[91,2] = PR[90,2] + -4.965;
   1:L PR[91] R[100]mm/sec CNT100;
   1:  PR[91,1] = PR[90,1] + 90.431;
   1:  PR[91,2] = PR[90,2] + -0.729;
   1:L PR[91] R[100]mm/sec CNT100;
   1:  PR[91,1] = PR[90,1] + 89.942;
   1:  PR[91,2] = PR[90,2] + 3.506;
   1:L PR[91] R[100]mm/sec CNT100;
   1:  PR[91,1] = PR[90,1] + 88.511;
   1:  PR[91,2] = PR[90,2] + 7.557;
   1:L PR[91] R[100]mm/sec CNT100;
   1:  PR[91,1] = PR[90,1] + 86.191;
   1:  PR[91,2] = PR[90,2] + 11.233;
   1:L PR[91] R[100]mm/sec CNT100;
   1:  PR[91,1] = PR[90,1] + 84.368;
   1:  PR[91,2] = PR[90,2] + 13.048;
   1:L PR[91] R[100]mm/sec CNT100;
   1:  PR[91,1] = PR[90,1] + 83.067;
   1:  PR[91,2] = PR[90,2] + 14.375;
   1:L PR[91] R[100]mm/sec CNT100;
   1:  PR[91,1] = PR[90,1] + 81.258;
   1:  PR[91,2] = PR[90,2] + 15.525;
   1:L PR[91] R[100]mm/sec CNT100;
   1:  PR[91,1] = PR[90,1] + 79.280;
   1:  PR[91,2] = PR[90,2] + 16.823;
   1:L PR[91] R[100]mm/sec CNT100;
   1:  PR[91,1] = PR[90,1] + 77.780;
   1:  PR[91,2] = PR[90,2] + 17.372;
   1:L PR[91] R[100]mm/sec CNT100;
   1:  PR[91,1] = PR[90,1] + 74.987;
   1:  PR[91,2] = PR[90,2] + 18.452;
   1:L PR[91] R[100]mm/sec CNT100;
   1:  PR[91,1] = PR[90,1] + 74.070;
   1:  PR[91,2] = PR[90,2] + 18.580;
   1:L PR[91] R[100]mm/sec CNT100;
   1:  PR[91,1] = PR[90,1] + 70.356;
   1:  PR[91,2] = PR[90,2] + 19.175;
   1:L PR[91] R[100]mm/sec CNT100;
   1:  PR[91,1] = PR[90,1] + 68.583;
   1:  PR[91,2] = PR[90,2] + 19.075;
   1:L PR[91] R[100]mm/sec CNT100;
   1:  PR[91,1] = PR[90,1] + 65.668;
   1:  PR[91,2] = PR[90,2] + 18.971;
   1:L PR[91] R[100]mm/sec CNT100;
   1:  PR[91,1] = PR[90,1] + 64.944;
   1:  PR[91,2] = PR[90,2] + 18.863;
   1:L PR[91] R[100]mm/sec CNT100;
   1:  PR[91,1] = PR[90,1] + 61.208;
   1:  PR[91,2] = PR[90,2] + 17.952;
   1:L PR[91] R[100]mm/sec CNT100;
   1:  PR[91,1] = PR[90,1] + 58.878;
   1:  PR[91,2] = PR[90,2] + 17.042;
   1:L PR[91] R[100]mm/sec CNT100;
   1:  PR[91,1] = PR[90,1] + 56.860;
   1:  PR[91,2] = PR[90,2] + 16.064;
   1:L PR[91] R[100]mm/sec CNT100;
   1:  PR[91,1] = PR[90,1] + 53.212;
   1:  PR[91,2] = PR[90,2] + 13.527;
   1:L PR[91] R[100]mm/sec CNT100;
   1:  PR[91,1] = PR[90,1] + 52.836;
   1:  PR[91,2] = PR[90,2] + 13.226;
   1:L PR[91] R[100]mm/sec CNT100;
   1:  PR[91,1] = PR[90,1] + 51.186;
   1:  PR[91,2] = PR[90,2] + 11.309;
   1:L PR[91] R[100]mm/sec CNT100;
   1:  PR[91,1] = PR[90,1] + 49.400;
   1:  PR[91,2] = PR[90,2] + 9.445;
   1:L PR[91] R[100]mm/sec CNT100;
   1:  PR[91,1] = PR[90,1] + 49.055;
   1:  PR[91,2] = PR[90,2] + 9.026;
   1:L PR[91] R[100]mm/sec CNT100;
   1:  PR[91,1] = PR[90,1] + 47.153;
   1:  PR[91,2] = PR[90,2] + 5.377;
   1:L PR[91] R[100]mm/sec CNT100;
   1:  PR[91,1] = PR[90,1] + 45.494;
   1:  PR[91,2] = PR[90,2] + -0.780;
   1:L PR[91] R[100]mm/sec CNT100TB   .50sec,CALL END_PUD;
   1:  PR[92] = PR[91];
   1:  PR[92,3] = PR[92,3] + 20;
   1:J PR[92] 10% FINE;
   1:  PR[91,1] = PR[90,1] + -2.545;
   1:  PR[91,2] = PR[90,2] + -5.813;
   1:  PR[92] = PR[91];
   1:  PR[92,3] = PR[92,3] + 20;
   1:J PR[92] 10% FINE;
   1:L PR[91] R[100]mm/sec CNT100;
   1:  CALL LASER_DRAHT_START;
   1:  PR[91,1] = PR[90,1] + -2.063;
   1:  PR[91,2] = PR[90,2] + -3.251;
   1:L PR[91] R[100]mm/sec CNT100;
   1:  PR[91,1] = PR[90,1] + -1.845;
   1:  PR[91,2] = PR[90,2] + -1.444;
   1:L PR[91] R[100]mm/sec CNT100;
   1:  PR[91,1] = PR[90,1] + -1.827;
   1:  PR[91,2] = PR[90,2] + -0.821;
   1:L PR[91] R[100]mm/sec CNT100;
   1:  PR[91,1] = PR[90,1] + -2.052;
   1:  PR[91,2] = PR[90,2] + 1.043;
   1:L PR[91] R[100]mm/sec CNT100;
   1:  PR[91,1] = PR[90,1] + -2.079;
   1:  PR[91,2] = PR[90,2] + 1.870;
   1:L PR[91] R[100]mm/sec CNT100;
   1:  PR[91,1] = PR[90,1] + -2.542;
   1:  PR[91,2] = PR[90,2] + 4.345;
   1:L PR[91] R[100]mm/sec CNT100;
   1:  PR[91,1] = PR[90,1] + -3.216;
   1:  PR[91,2] = PR[90,2] + 6.152;
   1:L PR[91] R[100]mm/sec CNT100;
   1:  PR[91,1] = PR[90,1] + -4.219;
   1:  PR[91,2] = PR[90,2] + 8.369;
   1:L PR[91] R[100]mm/sec CNT100;
   1:  PR[91,1] = PR[90,1] + -5.449;
   1:  PR[91,2] = PR[90,2] + 10.199;
   1:L PR[91] R[100]mm/sec CNT100;
   1:  PR[91,1] = PR[90,1] + -6.767;
   1:  PR[91,2] = PR[90,2] + 11.903;
   1:L PR[91] R[100]mm/sec CNT100;
   1:  PR[91,1] = PR[90,1] + -8.663;
   1:  PR[91,2] = PR[90,2] + 13.664;
   1:L PR[91] R[100]mm/sec CNT100;
   1:  PR[91,1] = PR[90,1] + -10.039;
   1:  PR[91,2] = PR[90,2] + 14.785;
   1:L PR[91] R[100]mm/sec CNT100;
   1:  PR[91,1] = PR[90,1] + -12.675;
   1:  PR[91,2] = PR[90,2] + 16.303;
   1:L PR[91] R[100]mm/sec CNT100;
   1:  PR[91,1] = PR[90,1] + -13.864;
   1:  PR[91,2] = PR[90,2] + 16.892;
   1:L PR[91] R[100]mm/sec CNT100;
   1:  PR[91,1] = PR[90,1] + -17.226;
   1:  PR[91,2] = PR[90,2] + 17.935;
   1:L PR[91] R[100]mm/sec CNT100;
   1:  PR[91,1] = PR[90,1] + -18.054;
   1:  PR[91,2] = PR[90,2] + 18.138;
   1:L PR[91] R[100]mm/sec CNT100;
   1:  PR[91,1] = PR[90,1] + -22.027;
   1:  PR[91,2] = PR[90,2] + 18.466;
   1:L PR[91] R[100]mm/sec CNT100;
   1:  PR[91,1] = PR[90,1] + -22.408;
   1:  PR[91,2] = PR[90,2] + 18.476;
   1:L PR[91] R[100]mm/sec CNT100;
   1:  PR[91,1] = PR[90,1] + -26.777;
   1:  PR[91,2] = PR[90,2] + 17.875;
   1:L PR[91] R[100]mm/sec CNT100;
   1:  PR[91,1] = PR[90,1] + -30.837;
   1:  PR[91,2] = PR[90,2] + 16.394;
   1:L PR[91] R[100]mm/sec CNT100;
   1:  PR[91,1] = PR[90,1] + -34.445;
   1:  PR[91,2] = PR[90,2] + 14.080;
   1:L PR[91] R[100]mm/sec CNT100;
   1:  PR[91,1] = PR[90,1] + -37.440;
   1:  PR[91,2] = PR[90,2] + 11.049;
   1:L PR[91] R[100]mm/sec CNT100;
   1:  PR[91,1] = PR[90,1] + -39.685;
   1:  PR[91,2] = PR[90,2] + 7.452;
   1:L PR[91] R[100]mm/sec CNT100;
   1:  PR[91,1] = PR[90,1] + -41.074;
   1:  PR[91,2] = PR[90,2] + 3.459;
   1:L PR[91] R[100]mm/sec CNT100;
   1:  PR[91,1] = PR[90,1] + -41.552;
   1:  PR[91,2] = PR[90,2] + -0.720;
   1:L PR[91] R[100]mm/sec CNT100;
   1:  PR[91,1] = PR[90,1] + -41.468;
   1:  PR[91,2] = PR[90,2] + -1.394;
   1:L PR[91] R[100]mm/sec CNT100;
   1:  PR[91,1] = PR[90,1] + -41.073;
   1:  PR[91,2] = PR[90,2] + -4.920;
   1:L PR[91] R[100]mm/sec CNT100;
   1:  PR[91,1] = PR[90,1] + -39.685;
   1:  PR[91,2] = PR[90,2] + -8.910;
   1:L PR[91] R[100]mm/sec CNT100;
   1:  PR[91,1] = PR[90,1] + -37.440;
   1:  PR[91,2] = PR[90,2] + -12.508;
   1:L PR[91] R[100]mm/sec CNT100;
   1:  PR[91,1] = PR[90,1] + -34.445;
   1:  PR[91,2] = PR[90,2] + -15.539;
   1:L PR[91] R[100]mm/sec CNT100;
   1:  PR[91,1] = PR[90,1] + -30.837;
   1:  PR[91,2] = PR[90,2] + -17.853;
   1:L PR[91] R[100]mm/sec CNT100;
   1:  PR[91,1] = PR[90,1] + -26.738;
   1:  PR[91,2] = PR[90,2] + -19.348;
   1:L PR[91] R[100]mm/sec CNT100;
   1:  PR[91,1] = PR[90,1] + -22.411;
   1:  PR[91,2] = PR[90,2] + -19.935;
   1:L PR[91] R[100]mm/sec CNT100;
   1:  PR[91,1] = PR[90,1] + -22.029;
   1:  PR[91,2] = PR[90,2] + -19.925;
   1:L PR[91] R[100]mm/sec CNT100;
   1:  PR[91,1] = PR[90,1] + -18.057;
   1:  PR[91,2] = PR[90,2] + -19.597;
   1:L PR[91] R[100]mm/sec CNT100;
   1:  PR[91,1] = PR[90,1] + -17.229;
   1:  PR[91,2] = PR[90,2] + -19.395;
   1:L PR[91] R[100]mm/sec CNT100;
   1:  PR[91,1] = PR[90,1] + -13.868;
   1:  PR[91,2] = PR[90,2] + -18.353;
   1:L PR[91] R[100]mm/sec CNT100;
   1:  PR[91,1] = PR[90,1] + -12.679;
   1:  PR[91,2] = PR[90,2] + -17.764;
   1:L PR[91] R[100]mm/sec CNT100;
   1:  PR[91,1] = PR[90,1] + -10.044;
   1:  PR[91,2] = PR[90,2] + -16.246;
   1:L PR[91] R[100]mm/sec CNT100;
   1:  PR[91,1] = PR[90,1] + -8.668;
   1:  PR[91,2] = PR[90,2] + -15.128;
   1:L PR[91] R[100]mm/sec CNT100;
   1:  PR[91,1] = PR[90,1] + -6.772;
   1:  PR[91,2] = PR[90,2] + -13.367;
   1:L PR[91] R[100]mm/sec CNT100;
   1:  PR[91,1] = PR[90,1] + -5.454;
   1:  PR[91,2] = PR[90,2] + -11.665;
   1:L PR[91] R[100]mm/sec CNT100;
   1:  PR[91,1] = PR[90,1] + -4.223;
   1:  PR[91,2] = PR[90,2] + -9.835;
   1:L PR[91] R[100]mm/sec CNT100;
   1:  PR[91,1] = PR[90,1] + -3.219;
   1:  PR[91,2] = PR[90,2] + -7.620;
   1:L PR[91] R[100]mm/sec CNT100;
   1:  PR[91,1] = PR[90,1] + -2.545;
   1:  PR[91,2] = PR[90,2] + -5.813;
   1:L PR[91] R[100]mm/sec CNT100TB   .50sec,CALL END_PUD;
   1:  PR[92] = PR[91];
   1:  PR[92,3] = PR[92,3] + 20;
   1:J PR[92] 10% FINE;
   1:  PR[91,1] = PR[90,1] + -49.402;
   1:  PR[91,2] = PR[90,2] + 2.907;
   1:  PR[92] = PR[91];
   1:  PR[92,3] = PR[92,3] + 20;
   1:J PR[92] 10% FINE;
   1:L PR[91] R[100]mm/sec CNT100;
   1:  CALL LASER_DRAHT_START;
   1:  PR[91,1] = PR[90,1] + -49.455;
   1:  PR[91,2] = PR[90,2] + 3.404;
   1:L PR[91] R[100]mm/sec CNT100;
   1:  PR[91,1] = PR[90,1] + -50.286;
   1:  PR[91,2] = PR[90,2] + 5.455;
   1:L PR[91] R[100]mm/sec CNT100;
   1:  PR[91,1] = PR[90,1] + -50.999;
   1:  PR[91,2] = PR[90,2] + 7.343;
   1:L PR[91] R[100]mm/sec CNT100;
   1:  PR[91,1] = PR[90,1] + -53.381;
   1:  PR[91,2] = PR[90,2] + 10.875;
   1:L PR[91] R[100]mm/sec CNT100;
   1:  PR[91,1] = PR[90,1] + -56.525;
   1:  PR[91,2] = PR[90,2] + 13.850;
   1:L PR[91] R[100]mm/sec CNT100;
   1:  PR[91,1] = PR[90,1] + -58.321;
   1:  PR[91,2] = PR[90,2] + 14.961;
   1:L PR[91] R[100]mm/sec CNT100;
   1:  PR[91,1] = PR[90,1] + -60.248;
   1:  PR[91,2] = PR[90,2] + 16.125;
   1:L PR[91] R[100]mm/sec CNT100;
   1:  PR[91,1] = PR[90,1] + -64.390;
   1:  PR[91,2] = PR[90,2] + 17.634;
   1:L PR[91] R[100]mm/sec CNT100;
   1:  PR[91,1] = PR[90,1] + -68.740;
   1:  PR[91,2] = PR[90,2] + 18.318;
   1:L PR[91] R[100]mm/sec CNT100;
   1:  PR[91,1] = PR[90,1] + -72.934;
   1:  PR[91,2] = PR[90,2] + 18.197;
   1:L PR[91] R[100]mm/sec CNT100;
   1:  PR[91,1] = PR[90,1] + -76.974;
   1:  PR[91,2] = PR[90,2] + 17.263;
   1:L PR[91] R[100]mm/sec CNT100;
   1:  PR[91,1] = PR[90,1] + -80.705;
   1:  PR[91,2] = PR[90,2] + 15.568;
   1:L PR[91] R[100]mm/sec CNT100;
   1:  PR[91,1] = PR[90,1] + -83.979;
   1:  PR[91,2] = PR[90,2] + 13.192;
   1:L PR[91] R[100]mm/sec CNT100;
   1:  PR[91,1] = PR[90,1] + -86.664;
   1:  PR[91,2] = PR[90,2] + 10.240;
   1:L PR[91] R[100]mm/sec CNT100;
   1:  PR[91,1] = PR[90,1] + -88.659;
   1:  PR[91,2] = PR[90,2] + 6.841;
   1:L PR[91] R[100]mm/sec CNT100;
   1:  PR[91,1] = PR[90,1] + -89.885;
   1:  PR[91,2] = PR[90,2] + 3.132;
   1:L PR[91] R[100]mm/sec CNT100;
   1:  PR[91,1] = PR[90,1] + -90.196;
   1:  PR[91,2] = PR[90,2] + 0.271;
   1:L PR[91] R[100]mm/sec CNT100;
   1:  PR[91,1] = PR[90,1] + -90.379;
   1:  PR[91,2] = PR[90,2] + -0.638;
   1:L PR[91] R[100]mm/sec CNT100;
   1:  PR[91,1] = PR[90,1] + -90.388;
   1:  PR[91,2] = PR[90,2] + -0.728;
   1:L PR[91] R[100]mm/sec CNT100;
   1:  PR[91,1] = PR[90,1] + -90.009;
   1:  PR[91,2] = PR[90,2] + -4.217;
   1:L PR[91] R[100]mm/sec CNT100;
   1:  PR[91,1] = PR[90,1] + -89.978;
   1:  PR[91,2] = PR[90,2] + -4.355;
   1:L PR[91] R[100]mm/sec CNT100;
   1:  PR[91,1] = PR[90,1] + -89.953;
   1:  PR[91,2] = PR[90,2] + -4.588;
   1:L PR[91] R[100]mm/sec CNT100;
   1:  PR[91,1] = PR[90,1] + -88.720;
   1:  PR[91,2] = PR[90,2] + -8.290;
   1:L PR[91] R[100]mm/sec CNT100;
   1:  PR[91,1] = PR[90,1] + -86.710;
   1:  PR[91,2] = PR[90,2] + -11.689;
   1:L PR[91] R[100]mm/sec CNT100;
   1:  PR[91,1] = PR[90,1] + -84.003;
   1:  PR[91,2] = PR[90,2] + -14.643;
   1:L PR[91] R[100]mm/sec CNT100;
   1:  PR[91,1] = PR[90,1] + -80.703;
   1:  PR[91,2] = PR[90,2] + -17.023;
   1:L PR[91] R[100]mm/sec CNT100;
   1:  PR[91,1] = PR[90,1] + -78.294;
   1:  PR[91,2] = PR[90,2] + -18.099;
   1:L PR[91] R[100]mm/sec CNT100;
   1:  PR[91,1] = PR[90,1] + -76.929;
   1:  PR[91,2] = PR[90,2] + -18.728;
   1:L PR[91] R[100]mm/sec CNT100;
   1:  PR[91,1] = PR[90,1] + -74.807;
   1:  PR[91,2] = PR[90,2] + -19.203;
   1:L PR[91] R[100]mm/sec CNT100;
   1:  PR[91,1] = PR[90,1] + -72.849;
   1:  PR[91,2] = PR[90,2] + -19.670;
   1:L PR[91] R[100]mm/sec CNT100;
   1:  PR[91,1] = PR[90,1] + -71.213;
   1:  PR[91,2] = PR[90,2] + -19.706;
   1:L PR[91] R[100]mm/sec CNT100;
   1:  PR[91,1] = PR[90,1] + -68.622;
   1:  PR[91,2] = PR[90,2] + -19.800;
   1:L PR[91] R[100]mm/sec CNT100;
   1:  PR[91,1] = PR[90,1] + -67.618;
   1:  PR[91,2] = PR[90,2] + -19.621;
   1:L PR[91] R[100]mm/sec CNT100;
   1:  PR[91,1] = PR[90,1] + -64.414;
   1:  PR[91,2] = PR[90,2] + -19.098;
   1:L PR[91] R[100]mm/sec CNT100;
   1:  PR[91,1] = PR[90,1] + -61.199;
   1:  PR[91,2] = PR[90,2] + -17.867;
   1:L PR[91] R[100]mm/sec CNT100;
   1:  PR[91,1] = PR[90,1] + -60.331;
   1:  PR[91,2] = PR[90,2] + -17.562;
   1:L PR[91] R[100]mm/sec CNT100;
   1:  PR[91,1] = PR[90,1] + -57.147;
   1:  PR[91,2] = PR[90,2] + -15.650;
   1:L PR[91] R[100]mm/sec CNT100;
   1:  PR[91,1] = PR[90,1] + -56.507;
   1:  PR[91,2] = PR[90,2] + -15.281;
   1:L PR[91] R[100]mm/sec CNT100;
   1:  PR[91,1] = PR[90,1] + -54.384;
   1:  PR[91,2] = PR[90,2] + -13.299;
   1:L PR[91] R[100]mm/sec CNT100;
   1:  PR[91,1] = PR[90,1] + -53.299;
   1:  PR[91,2] = PR[90,2] + -12.318;
   1:L PR[91] R[100]mm/sec CNT100;
   1:  PR[91,1] = PR[90,1] + -52.069;
   1:  PR[91,2] = PR[90,2] + -10.516;
   1:L PR[91] R[100]mm/sec CNT100;
   1:  PR[91,1] = PR[90,1] + -50.858;
   1:  PR[91,2] = PR[90,2] + -8.788;
   1:L PR[91] R[100]mm/sec CNT100;
   1:  PR[91,1] = PR[90,1] + -49.338;
   1:  PR[91,2] = PR[90,2] + -4.866;
   1:L PR[91] R[100]mm/sec CNT100;
   1:  PR[91,1] = PR[90,1] + -49.195;
   1:  PR[91,2] = PR[90,2] + -3.713;
   1:L PR[91] R[100]mm/sec CNT100;
   1:  PR[91,1] = PR[90,1] + -49.053;
   1:  PR[91,2] = PR[90,2] + -1.681;
   1:L PR[91] R[100]mm/sec CNT100;
   1:  PR[91,1] = PR[90,1] + -48.931;
   1:  PR[91,2] = PR[90,2] + -0.731;
   1:L PR[91] R[100]mm/sec CNT100;
   1:  PR[91,1] = PR[90,1] + -49.402;
   1:  PR[91,2] = PR[90,2] + 2.907;
   1:L PR[91] R[100]mm/sec CNT100TB   .50sec,CALL END_PUD;
   1:  PR[92] = PR[91];
   1:  PR[92,3] = PR[92,3] + 20;
   1:J PR[92] 10% FINE;
   1:  PR[91] = PR[90];
   1:  PR[91,1] = PR[90,1] + 69.952;
   1:  PR[91,2] = PR[90,2] + 19.345;
   1:  PR[91,3] = PR[90,3] + 35.295;
   1:  PR[92] = PR[91];
   1:  PR[92,3] = PR[92,3] + 20;
   1:J PR[92] 10% FINE;
   1:L PR[91] R[100]mm/sec CNT100;
   1:  CALL LASER_DRAHT_START;
   1:  PR[91,1] = PR[90,1] + 69.657;
   1:  PR[91,2] = PR[90,2] + 19.366;
   1:L PR[91] R[100]mm/sec CNT100;
   1:  PR[91,1] = PR[90,1] + 65.452;
   1:  PR[91,2] = PR[90,2] + 19.215;
   1:L PR[91] R[100]mm/sec CNT100;
   1:  PR[91,1] = PR[90,1] + 63.586;
   1:  PR[91,2] = PR[90,2] + 18.937;
   1:L PR[91] R[100]mm/sec CNT100;
   1:  PR[91,1] = PR[90,1] + 60.886;
   1:  PR[91,2] = PR[90,2] + 18.279;
   1:L PR[91] R[100]mm/sec CNT100;
   1:  PR[91,1] = PR[90,1] + 57.334;
   1:  PR[91,2] = PR[90,2] + 16.892;
   1:L PR[91] R[100]mm/sec CNT100;
   1:  PR[91,1] = PR[90,1] + 56.403;
   1:  PR[91,2] = PR[90,2] + 16.440;
   1:L PR[91] R[100]mm/sec CNT100;
   1:  PR[91,1] = PR[90,1] + 53.336;
   1:  PR[91,2] = PR[90,2] + 14.308;
   1:L PR[91] R[100]mm/sec CNT100;
   1:  PR[91,1] = PR[90,1] + 52.055;
   1:  PR[91,2] = PR[90,2] + 13.518;
   1:L PR[91] R[100]mm/sec CNT100;
   1:  PR[91,1] = PR[90,1] + 51.768;
   1:  PR[91,2] = PR[90,2] + 13.306;
   1:L PR[91] R[100]mm/sec CNT100;
   1:  PR[91,1] = PR[90,1] + 48.909;
   1:  PR[91,2] = PR[90,2] + 10.322;
   1:L PR[91] R[100]mm/sec CNT100;
   1:  PR[91,1] = PR[90,1] + 47.681;
   1:  PR[91,2] = PR[90,2] + 8.831;
   1:L PR[91] R[100]mm/sec CNT100;
   1:  PR[91,1] = PR[90,1] + 46.544;
   1:  PR[91,2] = PR[90,2] + 6.639;
   1:L PR[91] R[100]mm/sec CNT100;
   1:  PR[91,1] = PR[90,1] + 44.305;
   1:  PR[91,2] = PR[90,2] + 2.562;
   1:L PR[91] R[100]mm/sec CNT100;
   1:  PR[91,1] = PR[90,1] + 41.592;
   1:  PR[91,2] = PR[90,2] + 8.703;
   1:L PR[91] R[100]mm/sec CNT100;
   1:  PR[91,1] = PR[90,1] + 41.274;
   1:  PR[91,2] = PR[90,2] + 9.287;
   1:L PR[91] R[100]mm/sec CNT100;
